LIN {X 0,Y 516.896,Z 484.102,A -85,B 0,C 180,E1 -5072.543,E2 -5072.543} C_VEL
LIN {X 0,Y 516.867,Z 484.105,A -85,B 0,C 180,E1 -5075.329,E2 -5075.329} C_VEL
LIN {X 0,Y 516.881,Z 484.098,A -85,B 0,C 180,E1 -5077.943,E2 -5077.943} C_VEL
LIN {X 0,Y 516.885,Z 484.1,A -85,B 0,C 180,E1 -5080.742,E2 -5080.742} C_VEL
LIN {X 0,Y 516.884,Z 484.103,A -85,B 0,C 180,E1 -5082.831,E2 -5082.831} C_VEL
LIN {X 0,Y 516.897,Z 484.096,A -85,B 0,C 180,E1 -5085.007,E2 -5085.007} C_VEL
LIN {X 0,Y 516.916,Z 484.093,A -85,B 0,C 180,E1 -5088.399,E2 -5088.399} C_VEL
LIN {X 0,Y 516.884,Z 484.143,A -85,B 0,C 180,E1 -5091.046,E2 -5091.046} C_VEL
LIN {X 0,Y 518.914,Z 494.433,A -85,B 0,C 180,E1 -5093.663,E2 -5093.663} C_VEL
LIN {X 0,Y 518.765,Z 503.318,A -85,B 0,C 180,E1 -5095.731,E2 -5095.731} C_VEL
LIN {X 0,Y 518.365,Z 517.844,A -85,B 0,C 180,E1 -5098.989,E2 -5098.989} C_VEL
LIN {X 0,Y 518.058,Z 531.109,A -85,B 0,C 180,E1 -5101.86,E2 -5101.86} C_VEL
LIN {X 0,Y 517.746,Z 545.538,A -85,B 0,C 180,E1 -5104.9,E2 -5104.9} C_VEL
LIN {X 0,Y 517.484,Z 558.916,A -85,B 0,C 180,E1 -5107.65,E2 -5107.65} C_VEL
LIN {X 0,Y 517.263,Z 573.383,A -85,B 0,C 180,E1 -5110.556,E2 -5110.556} C_VEL
LIN {X 0,Y 517.038,Z 587.913,A -85,B 0,C 180,E1 -5113.414,E2 -5113.414} C_VEL
LIN {X 0,Y 516.818,Z 601.396,A -85,B 0,C 180,E1 -5116.057,E2 -5116.057} C_VEL
LIN {X 0,Y 518.532,Z 613.647,A -85,B 0,C 180,E1 -5116.354,E2 -5116.354} C_VEL
LIN {X 0,Y 518.297,Z 626.806,A -85,B 0,C 180,E1 -5116.772,E2 -5116.772} C_VEL
LIN {X 0,Y 518.011,Z 637.948,A -85,B 0,C 180,E1 -5117.263,E2 -5117.263} C_VEL
LIN {X 0,Y 517.786,Z 649.556,A -85,B 0,C 180,E1 -5117.927,E2 -5117.927} C_VEL
LIN {X 0,Y 517.451,Z 660.748,A -85,B 0,C 180,E1 -5118.741,E2 -5118.741} C_VEL
LIN {X 0,Y 517.174,Z 670.566,A -85,B 0,C 180,E1 -5119.627,E2 -5119.627} C_VEL
LIN {X 0,Y 516.898,Z 679.413,A -85,B 0,C 180,E1 -5120.61,E2 -5120.61} C_VEL
LIN {X 0,Y 516.682,Z 688.004,A -85,B 0,C 180,E1 -5121.789,E2 -5121.789} C_VEL
LIN {X 0,Y 516.506,Z 694.868,A -85,B 0,C 180,E1 -5122.966,E2 -5122.966} C_VEL
LIN {X 0,Y 516.454,Z 700.366,A -85,B 0,C 180,E1 -5124.142,E2 -5124.142} C_VEL
LIN {X 0,Y 516.271,Z 704.677,A -85,B 0,C 180,E1 -5125.315,E2 -5125.315} C_VEL
LIN {X 0,Y 516.355,Z 706.958,A -85,B 0,C 180,E1 -5126.098,E2 -5126.098} C_VEL
LIN {X 0,Y 516.282,Z 708.807,A -85,B 0,C 180,E1 -5126.879,E2 -5126.879} C_VEL
LIN {X 0,Y 516.261,Z 710.193,A -85,B 0,C 180,E1 -5127.659,E2 -5127.659} C_VEL
LIN {X 0,Y 516.16,Z 711.785,A -85,B 0,C 180,E1 -5129.22,E2 -5129.22} C_VEL
LIN {X 0,Y 516.154,Z 712,A -85,B 0,C 180,E1 -5130,E2 -5130} C_VEL
LIN {X 0,Y 516.192,Z 711.183,A -85,B 0,C 180,E1 -5131.56,E2 -5131.56} C_VEL
LIN {X 0,Y 516.261,Z 710.196,A -85,B 0,C 180,E1 -5132.341,E2 -5132.341} C_VEL
LIN {X 0,Y 516.282,Z 708.81,A -85,B 0,C 180,E1 -5133.121,E2 -5133.121} C_VEL
LIN {X 0,Y 516.344,Z 705.895,A -85,B 0,C 180,E1 -5134.293,E2 -5134.293} C_VEL
LIN {X 0,Y 516.405,Z 701.947,A -85,B 0,C 180,E1 -5135.467,E2 -5135.467} C_VEL
LIN {X 0,Y 516.486,Z 696.032,A -85,B 0,C 180,E1 -5136.808,E2 -5136.808} C_VEL
LIN {X 0,Y 516.641,Z 689.234,A -85,B 0,C 180,E1 -5138.015,E2 -5138.015} C_VEL
LIN {X 0,Y 516.868,Z 680.991,A -85,B 0,C 180,E1 -5139.194,E2 -5139.194} C_VEL
LIN {X 0,Y 517.081,Z 672.519,A -85,B 0,C 180,E1 -5140.177,E2 -5140.177} C_VEL
LIN {X 0,Y 517.408,Z 661.937,A -85,B 0,C 180,E1 -5141.161,E2 -5141.161} C_VEL
LIN {X 0,Y 517.723,Z 650.028,A -85,B 0,C 180,E1 -5142.04,E2 -5142.04} C_VEL
LIN {X 0,Y 518.043,Z 637.865,A -85,B 0,C 180,E1 -5142.736,E2 -5142.736} C_VEL
LIN {X 0,Y 518.338,Z 625.358,A -85,B 0,C 180,E1 -5143.277,E2 -5143.277} C_VEL
LIN {X 0,Y 518.376,Z 612.02,A -85,B 0,C 180,E1 -5143.688,E2 -5143.688} C_VEL
LIN {X 0,Y 516.818,Z 601.178,A -85,B 0,C 180,E1 -5143.943,E2 -5143.943} C_VEL
LIN {X 0,Y 517.097,Z 584.267,A -85,B 0,C 180,E1 -5147.194,E2 -5147.194} C_VEL
LIN {X 0,Y 517.248,Z 569.103,A -85,B 0,C 180,E1 -5150.113,E2 -5150.113} C_VEL
LIN {X 0,Y 517.442,Z 555.28,A -85,B 0,C 180,E1 -5152.825,E2 -5152.825} C_VEL
LIN {X 0,Y 517.604,Z 541.77,A -85,B 0,C 180,E1 -5155.538,E2 -5155.538} C_VEL
LIN {X 0,Y 517.8,Z 526.86,A -85,B 0,C 180,E1 -5158.584,E2 -5158.584} C_VEL
LIN {X 0,Y 517.993,Z 512.786,A -85,B 0,C 180,E1 -5161.562,E2 -5161.562} C_VEL
LIN {X 0,Y 518.272,Z 498.486,A -85,B 0,C 180,E1 -5164.718,E2 -5164.718} C_VEL
LIN {X 0,Y 518.362,Z 492.293,A -85,B 0,C 180,E1 -5166.142,E2 -5166.142} C_VEL
LIN {X 0,Y 516.897,Z 484.1,A -85,B 0,C 180,E1 -5168.246,E2 -5168.246} C_VEL
LIN {X 0,Y 516.918,Z 484.098,A -85,B 0,C 180,E1 -5171.602,E2 -5171.602} C_VEL
LIN {X 0,Y 516.926,Z 484.1,A -85,B 0,C 180,E1 -5175.01,E2 -5175.01} C_VEL
LIN {X 0,Y 516.919,Z 484.099,A -85,B 0,C 180,E1 -5178.399,E2 -5178.399} C_VEL
LIN {X 0,Y 516.883,Z 484.102,A -85,B 0,C 180,E1 -5181.284,E2 -5181.284} C_VEL
LIN {X 0,Y 516.871,Z 484.102,A -85,B 0,C 180,E1 -5184.22,E2 -5184.22} C_VEL
LIN {X 0,Y 516.884,Z 484.101,A -85,B 0,C 180,E1 -5187.052,E2 -5187.052} C_VEL
LIN {X 0,Y 516.896,Z 484.101,A -85,B 0,C 180,E1 -5189.797,E2 -5189.797} C_VEL
LIN {X 0,Y 516.928,Z 484.096,A -85,B 0,C 180,E1 -5192.467,E2 -5192.467} C_VEL
LIN {X 0,Y 516.876,Z 484.102,A -85,B 0,C 180,E1 -5195.07,E2 -5195.07} C_VEL
LIN {X 0,Y 516.873,Z 484.102,A -85,B 0,C 180,E1 -5197.622,E2 -5197.622} C_VEL
LIN {X 0,Y 516.936,Z 484.095,A -85,B 0,C 180,E1 -5200.13,E2 -5200.13} C_VEL
LIN {X 0,Y 516.91,Z 484.098,A -85,B 0,C 180,E1 -5202.596,E2 -5202.596} C_VEL
LIN {X 0,Y 516.945,Z 484.092,A -85,B 0,C 180,E1 -5205.03,E2 -5205.03} C_VEL
LIN {X 0,Y 516.971,Z 484.09,A -85,B 0,C 180,E1 -5208.234,E2 -5208.234} C_VEL
LIN {X 0,Y 516.969,Z 484.088,A -85,B 0,C 180,E1 -5211.4,E2 -5211.4} C_VEL
LIN {X 0,Y 517.016,Z 484.085,A -85,B 0,C 180,E1 -5213.757,E2 -5213.757} C_VEL
LIN {X 0,Y 517.085,Z 484.075,A -85,B 0,C 180,E1 -5217.663,E2 -5217.663} C_VEL
LIN {X 0,Y 517.097,Z 484.075,A -85,B 0,C 180,E1 -5220.779,E2 -5220.779} C_VEL
LIN {X 0,Y 517.014,Z 484.085,A -85,B 0,C 180,E1 -5223.117,E2 -5223.117} C_VEL
LIN {X 0,Y 516.98,Z 484.088,A -85,B 0,C 180,E1 -5226.244,E2 -5226.244} C_VEL
LIN {X 0,Y 516.97,Z 484.09,A -85,B 0,C 180,E1 -5228.601,E2 -5228.601} C_VEL
LIN {X 0,Y 516.957,Z 484.092,A -85,B 0,C 180,E1 -5231.807,E2 -5231.807} C_VEL
LIN {X 0,Y 516.95,Z 484.093,A -85,B 0,C 180,E1 -5235.147,E2 -5235.147} C_VEL
LIN {X 0,Y 516.922,Z 484.101,A -85,B 0,C 180,E1 -5238.223,E2 -5238.223} C_VEL
LIN {X 0,Y 516.961,Z 484.207,A -85,B 0,C 180,E1 -5240.934,E2 -5240.934} C_VEL
LIN {X 0,Y 518.09,Z 488.502,A -85,B 0,C 180,E1 -5241.173,E2 -5241.173} C_VEL
LIN {X 0,Y 518.099,Z 498.056,A -85,B 0,C 180,E1 -5241.694,E2 -5241.694} C_VEL
LIN {X 0,Y 517.842,Z 508.776,A -85,B 0,C 180,E1 -5242.422,E2 -5242.422} C_VEL
LIN {X 0,Y 517.549,Z 518.004,A -85,B 0,C 180,E1 -5243.192,E2 -5243.192} C_VEL
LIN {X 0,Y 517.283,Z 526.537,A -85,B 0,C 180,E1 -5244.054,E2 -5244.054} C_VEL
LIN {X 0,Y 516.981,Z 535.368,A -85,B 0,C 180,E1 -5245.14,E2 -5245.14} C_VEL
LIN {X 0,Y 516.804,Z 543.287,A -85,B 0,C 180,E1 -5246.365,E2 -5246.365} C_VEL
LIN {X 0,Y 516.615,Z 549.379,A -85,B 0,C 180,E1 -5247.551,E2 -5247.551} C_VEL
LIN {X 0,Y 516.501,Z 553.171,A -85,B 0,C 180,E1 -5248.441,E2 -5248.441} C_VEL
LIN {X 0,Y 516.423,Z 557.58,A -85,B 0,C 180,E1 -5249.791,E2 -5249.791} C_VEL
LIN {X 0,Y 516.345,Z 560.715,A -85,B 0,C 180,E1 -5251.146,E2 -5251.146} C_VEL
LIN {X 0,Y 516.265,Z 562.567,A -85,B 0,C 180,E1 -5252.433,E2 -5252.433} C_VEL
LIN {X 0,Y 516.287,Z 563.411,A -85,B 0,C 180,E1 -5253.926,E2 -5253.926} C_VEL
LIN {X 0,Y 516.253,Z 562.97,A -85,B 0,C 180,E1 -5255.233,E2 -5255.233} C_VEL
LIN {X 0,Y 516.3,Z 560.93,A -85,B 0,C 180,E1 -5256.794,E2 -5256.794} C_VEL
LIN {X 0,Y 516.412,Z 558.616,A -85,B 0,C 180,E1 -5257.876,E2 -5257.876} C_VEL
LIN {X 0,Y 516.47,Z 554.854,A -85,B 0,C 180,E1 -5259.136,E2 -5259.136} C_VEL
LIN {X 0,Y 516.54,Z 551.346,A -85,B 0,C 180,E1 -5260.061,E2 -5260.061} C_VEL
LIN {X 0,Y 516.649,Z 546.133,A -85,B 0,C 180,E1 -5261.168,E2 -5261.168} C_VEL
LIN {X 0,Y 516.811,Z 541.161,A -85,B 0,C 180,E1 -5262.048,E2 -5262.048} C_VEL
LIN {X 0,Y 517.041,Z 534.094,A -85,B 0,C 180,E1 -5263.082,E2 -5263.082} C_VEL
LIN {X 0,Y 517.207,Z 527.215,A -85,B 0,C 180,E1 -5263.93,E2 -5263.93} C_VEL
LIN {X 0,Y 517.478,Z 518.829,A -85,B 0,C 180,E1 -5264.792,E2 -5264.792} C_VEL
LIN {X 0,Y 517.631,Z 513.549,A -85,B 0,C 180,E1 -5265.266,E2 -5265.266} C_VEL
LIN {X 0,Y 517.058,Z 507.251,A -85,B 0,C 180,E1 -5265.784,E2 -5265.784} C_VEL
LIN {X 0,Y 515.311,Z 500.945,A -85,B 0,C 180,E1 -5266.275,E2 -5266.275} C_VEL
LIN {X 0,Y 513.049,Z 494.539,A -85,B 0,C 180,E1 -5266.742,E2 -5266.742} C_VEL
LIN {X 0,Y 510.614,Z 487.934,A -85,B 0,C 180,E1 -5267.163,E2 -5267.163} C_VEL
LIN {X 0,Y 509.873,Z 484.974,A -85,B 0,C 180,E1 -5267.337,E2 -5267.337} C_VEL
LIN {X 0,Y 509.842,Z 484.979,A -85,B 0,C 180,E1 -5270.647,E2 -5270.647} C_VEL
LIN {X 0,Y 509.814,Z 484.982,A -85,B 0,C 180,E1 -5273.646,E2 -5273.646} C_VEL
LIN {X 0,Y 509.864,Z 484.974,A -85,B 0,C 180,E1 -5276.539,E2 -5276.539} C_VEL
LIN {X 0,Y 509.846,Z 484.976,A -85,B 0,C 180,E1 -5279.334,E2 -5279.334} C_VEL
LIN {X 0,Y 509.891,Z 484.97,A -85,B 0,C 180,E1 -5282.054,E2 -5282.054} C_VEL
LIN {X 0,Y 509.823,Z 484.981,A -85,B 0,C 180,E1 -5284.701,E2 -5284.701} C_VEL
LIN {X 0,Y 509.832,Z 484.982,A -85,B 0,C 180,E1 -5287.458,E2 -5287.458} C_VEL
LIN {X 0,Y 509.922,Z 484.967,A -85,B 0,C 180,E1 -5289.845,E2 -5289.845} C_VEL
LIN {X 0,Y 509.872,Z 484.975,A -85,B 0,C 180,E1 -5293.174,E2 -5293.174} C_VEL
LIN {X 0,Y 509.863,Z 484.974,A -85,B 0,C 180,E1 -5295.634,E2 -5295.634} C_VEL
LIN {X 0,Y 509.919,Z 484.967,A -85,B 0,C 180,E1 -5298.874,E2 -5298.874} C_VEL
LIN {X 0,Y 509.915,Z 484.97,A -85,B 0,C 180,E1 -5302.078,E2 -5302.078} C_VEL
LIN {X 0,Y 509.97,Z 484.96,A -85,B 0,C 180,E1 -5304.464,E2 -5304.464} C_VEL
LIN {X 0,Y 510.06,Z 484.949,A -85,B 0,C 180,E1 -5307.631,E2 -5307.631} C_VEL
LIN {X 0,Y 510.067,Z 484.948,A -85,B 0,C 180,E1 -5310.789,E2 -5310.789} C_VEL
LIN {X 0,Y 509.933,Z 484.967,A -85,B 0,C 180,E1 -5313.16,E2 -5313.16} C_VEL
LIN {X 0,Y 509.927,Z 484.966,A -85,B 0,C 180,E1 -5316.33,E2 -5316.33} C_VEL
LIN {X 0,Y 509.916,Z 484.969,A -85,B 0,C 180,E1 -5318.72,E2 -5318.72} C_VEL
LIN {X 0,Y 509.91,Z 484.97,A -85,B 0,C 180,E1 -5321.931,E2 -5321.931} C_VEL
LIN {X 0,Y 509.9,Z 484.97,A -85,B 0,C 180,E1 -5325.242,E2 -5325.242} C_VEL
LIN {X 0,Y 509.862,Z 484.973,A -85,B 0,C 180,E1 -5328.484,E2 -5328.484} C_VEL
LIN {X 0,Y 509.856,Z 484.978,A -85,B 0,C 180,E1 -5331.001,E2 -5331.001} C_VEL
LIN {X 0,Y 509.824,Z 484.982,A -85,B 0,C 180,E1 -5333.564,E2 -5333.564} C_VEL
LIN {X 0,Y 509.882,Z 484.972,A -85,B 0,C 180,E1 -5336.37,E2 -5336.37} C_VEL
LIN {X 0,Y 509.863,Z 484.977,A -85,B 0,C 180,E1 -5339.726,E2 -5339.726} C_VEL
LIN {X 0,Y 509.871,Z 484.976,A -85,B 0,C 180,E1 -5342.773,E2 -5342.773} C_VEL
LIN {X 0,Y 509.826,Z 484.982,A -85,B 0,C 180,E1 -5345.577,E2 -5345.577} C_VEL
LIN {X 0,Y 509.853,Z 484.975,A -85,B 0,C 180,E1 -5348.338,E2 -5348.338} C_VEL
LIN {X 0,Y 509.836,Z 484.979,A -85,B 0,C 180,E1 -5351.428,E2 -5351.428} C_VEL
LIN {X 0,Y 509.843,Z 484.979,A -85,B 0,C 180,E1 -5354.67,E2 -5354.67} C_VEL
LIN {X 0,Y 509.853,Z 484.976,A -85,B 0,C 180,E1 -5358.104,E2 -5358.104} C_VEL
LIN {X 0,Y 509.849,Z 484.978,A -85,B 0,C 180,E1 -5360.647,E2 -5360.647} C_VEL
LIN {X 0,Y 509.809,Z 484.984,A -85,B 0,C 180,E1 -5363.645,E2 -5363.645} C_VEL
LIN {X 0,Y 509.863,Z 484.976,A -85,B 0,C 180,E1 -5366.539,E2 -5366.539} C_VEL
LIN {X 0,Y 509.849,Z 484.977,A -85,B 0,C 180,E1 -5369.334,E2 -5369.334} C_VEL
LIN {X 0,Y 509.895,Z 484.969,A -85,B 0,C 180,E1 -5372.054,E2 -5372.054} C_VEL
LIN {X 0,Y 509.82,Z 484.98,A -85,B 0,C 180,E1 -5374.701,E2 -5374.701} C_VEL
LIN {X 0,Y 509.83,Z 484.979,A -85,B 0,C 180,E1 -5377.458,E2 -5377.458} C_VEL
LIN {X 0,Y 509.918,Z 484.969,A -85,B 0,C 180,E1 -5379.844,E2 -5379.844} C_VEL
LIN {X 0,Y 509.873,Z 484.976,A -85,B 0,C 180,E1 -5383.174,E2 -5383.174} C_VEL
LIN {X 0,Y 509.862,Z 484.975,A -85,B 0,C 180,E1 -5385.634,E2 -5385.634} C_VEL
LIN {X 0,Y 509.917,Z 484.969,A -85,B 0,C 180,E1 -5388.874,E2 -5388.874} C_VEL
LIN {X 0,Y 509.911,Z 484.97,A -85,B 0,C 180,E1 -5392.078,E2 -5392.078} C_VEL
LIN {X 0,Y 509.975,Z 484.96,A -85,B 0,C 180,E1 -5394.464,E2 -5394.464} C_VEL
LIN {X 0,Y 510.053,Z 484.951,A -85,B 0,C 180,E1 -5397.631,E2 -5397.631} C_VEL
LIN {X 0,Y 510.066,Z 484.95,A -85,B 0,C 180,E1 -5400.789,E2 -5400.789} C_VEL
LIN {X 0,Y 509.919,Z 484.967,A -85,B 0,C 180,E1 -5403.16,E2 -5403.16} C_VEL
LIN {X 0,Y 509.928,Z 484.965,A -85,B 0,C 180,E1 -5406.33,E2 -5406.33} C_VEL
LIN {X 0,Y 509.913,Z 484.971,A -85,B 0,C 180,E1 -5408.72,E2 -5408.72} C_VEL
LIN {X 0,Y 509.955,Z 484.964,A -85,B 0,C 180,E1 -5411.93,E2 -5411.93} C_VEL
LIN {X 0,Y 509.897,Z 484.97,A -85,B 0,C 180,E1 -5415.242,E2 -5415.242} C_VEL
LIN {X 0,Y 509.864,Z 484.974,A -85,B 0,C 180,E1 -5418.484,E2 -5418.484} C_VEL
LIN {X 0,Y 509.852,Z 484.976,A -85,B 0,C 180,E1 -5421.002,E2 -5421.002} C_VEL
LIN {X 0,Y 509.823,Z 484.981,A -85,B 0,C 180,E1 -5423.564,E2 -5423.564} C_VEL
LIN {X 0,Y 509.875,Z 484.974,A -85,B 0,C 180,E1 -5426.37,E2 -5426.37} C_VEL
LIN {X 0,Y 509.86,Z 484.976,A -85,B 0,C 180,E1 -5429.726,E2 -5429.726} C_VEL
LIN {X 0,Y 509.868,Z 484.975,A -85,B 0,C 180,E1 -5432.773,E2 -5432.773} C_VEL
LIN {X 0,Y 509.827,Z 484.981,A -85,B 0,C 180,E1 -5435.578,E2 -5435.578} C_VEL
LIN {X 0,Y 509.85,Z 484.977,A -85,B 0,C 180,E1 -5438.338,E2 -5438.338} C_VEL
LIN {X 0,Y 509.857,Z 484.979,A -85,B 0,C 180,E1 -5441.425,E2 -5441.425} C_VEL
LIN {X 0,Y 509.84,Z 484.977,A -85,B 0,C 180,E1 -5444.67,E2 -5444.67} C_VEL
LIN {X 0,Y 509.856,Z 484.972,A -85,B 0,C 180,E1 -5448.104,E2 -5448.104} C_VEL
LIN {X 0,Y 509.847,Z 485.024,A -85,B 0,C 180,E1 -5450.775,E2 -5450.775} C_VEL
LIN {X 0,Y 511.835,Z 494.949,A -85,B 0,C 180,E1 -5453.346,E2 -5453.346} C_VEL
LIN {X 0,Y 512.044,Z 497.933,A -85,B 0,C 180,E1 -5454.076,E2 -5454.076} C_VEL
LIN {X 0,Y 511.677,Z 509.084,A -85,B 0,C 180,E1 -5456.673,E2 -5456.673} C_VEL
LIN {X 0,Y 511.292,Z 523.821,A -85,B 0,C 180,E1 -5459.994,E2 -5459.994} C_VEL
LIN {X 0,Y 510.931,Z 537.675,A -85,B 0,C 180,E1 -5463.004,E2 -5463.004} C_VEL
LIN {X 0,Y 510.624,Z 552.005,A -85,B 0,C 180,E1 -5466.045,E2 -5466.045} C_VEL
LIN {X 0,Y 510.26,Z 567.756,A -85,B 0,C 180,E1 -5469.297,E2 -5469.297} C_VEL
LIN {X 0,Y 510.057,Z 582.932,A -85,B 0,C 180,E1 -5472.354,E2 -5472.354} C_VEL
LIN {X 0,Y 509.79,Z 599.301,A -85,B 0,C 180,E1 -5475.632,E2 -5475.632} C_VEL
LIN {X 0,Y 509.8,Z 600.447,A -85,B 0,C 180,E1 -5475.862,E2 -5475.862} C_VEL
LIN {X 0,Y 510.811,Z 608.526,A -85,B 0,C 180,E1 -5476.049,E2 -5476.049} C_VEL
LIN {X 0,Y 511.563,Z 615.375,A -85,B 0,C 180,E1 -5476.241,E2 -5476.241} C_VEL
LIN {X 0,Y 511.287,Z 628.315,A -85,B 0,C 180,E1 -5476.689,E2 -5476.689} C_VEL
LIN {X 0,Y 510.934,Z 640.657,A -85,B 0,C 180,E1 -5477.286,E2 -5477.286} C_VEL
LIN {X 0,Y 510.637,Z 651.496,A -85,B 0,C 180,E1 -5477.962,E2 -5477.962} C_VEL
LIN {X 0,Y 510.336,Z 662.111,A -85,B 0,C 180,E1 -5478.783,E2 -5478.783} C_VEL
LIN {X 0,Y 510.061,Z 671.583,A -85,B 0,C 180,E1 -5479.681,E2 -5479.681} C_VEL
LIN {X 0,Y 509.802,Z 680.238,A -85,B 0,C 180,E1 -5480.678,E2 -5480.678} C_VEL
LIN {X 0,Y 509.585,Z 688.692,A -85,B 0,C 180,E1 -5481.873,E2 -5481.873} C_VEL
LIN {X 0,Y 509.42,Z 695.519,A -85,B 0,C 180,E1 -5483.067,E2 -5483.067} C_VEL
LIN {X 0,Y 509.322,Z 701.779,A -85,B 0,C 180,E1 -5484.457,E2 -5484.457} C_VEL
LIN {X 0,Y 509.232,Z 705.811,A -85,B 0,C 180,E1 -5485.647,E2 -5485.647} C_VEL
LIN {X 0,Y 509.2,Z 708.77,A -85,B 0,C 180,E1 -5486.835,E2 -5486.835} C_VEL
LIN {X 0,Y 509.161,Z 710.171,A -85,B 0,C 180,E1 -5487.627,E2 -5487.627} C_VEL
LIN {X 0,Y 509.073,Z 711.774,A -85,B 0,C 180,E1 -5489.209,E2 -5489.209} C_VEL
LIN {X 0,Y 509.065,Z 711.991,A -85,B 0,C 180,E1 -5490,E2 -5490} C_VEL
LIN {X 0,Y 509.112,Z 711.169,A -85,B 0,C 180,E1 -5491.582,E2 -5491.582} C_VEL
LIN {X 0,Y 509.161,Z 710.174,A -85,B 0,C 180,E1 -5492.373,E2 -5492.373} C_VEL
LIN {X 0,Y 509.2,Z 708.774,A -85,B 0,C 180,E1 -5493.165,E2 -5493.165} C_VEL
LIN {X 0,Y 509.232,Z 705.812,A -85,B 0,C 180,E1 -5494.353,E2 -5494.353} C_VEL
LIN {X 0,Y 509.322,Z 701.776,A -85,B 0,C 180,E1 -5495.543,E2 -5495.543} C_VEL
LIN {X 0,Y 509.405,Z 695.97,A -85,B 0,C 180,E1 -5496.844,E2 -5496.844} C_VEL
LIN {X 0,Y 509.585,Z 688.657,A -85,B 0,C 180,E1 -5498.127,E2 -5498.127} C_VEL
LIN {X 0,Y 509.802,Z 680.168,A -85,B 0,C 180,E1 -5499.322,E2 -5499.322} C_VEL
LIN {X 0,Y 510.061,Z 671.474,A -85,B 0,C 180,E1 -5500.319,E2 -5500.319} C_VEL
LIN {X 0,Y 510.364,Z 660.755,A -85,B 0,C 180,E1 -5501.317,E2 -5501.317} C_VEL
LIN {X 0,Y 510.671,Z 649.828,A -85,B 0,C 180,E1 -5502.139,E2 -5502.139} C_VEL
LIN {X 0,Y 511.003,Z 638.603,A -85,B 0,C 180,E1 -5502.813,E2 -5502.813} C_VEL
LIN {X 0,Y 511.319,Z 626.732,A -85,B 0,C 180,E1 -5503.361,E2 -5503.361} C_VEL
LIN {X 0,Y 511.473,Z 613.096,A -85,B 0,C 180,E1 -5503.813,E2 -5503.813} C_VEL
LIN {X 0,Y 509.848,Z 601.602,A -85,B 0,C 180,E1 -5504.099,E2 -5504.099} C_VEL
LIN {X 0,Y 509.791,Z 599.936,A -85,B 0,C 180,E1 -5504.164,E2 -5504.164} C_VEL
LIN {X 0,Y 510.007,Z 584.216,A -85,B 0,C 180,E1 -5507.234,E2 -5507.234} C_VEL
LIN {X 0,Y 510.165,Z 569.301,A -85,B 0,C 180,E1 -5510.145,E2 -5510.145} C_VEL
LIN {X 0,Y 510.385,Z 554.534,A -85,B 0,C 180,E1 -5513.107,E2 -5513.107} C_VEL
LIN {X 0,Y 510.583,Z 540.738,A -85,B 0,C 180,E1 -5515.915,E2 -5515.915} C_VEL
LIN {X 0,Y 510.803,Z 525.911,A -85,B 0,C 180,E1 -5519.012,E2 -5519.012} C_VEL
LIN {X 0,Y 511.056,Z 512.231,A -85,B 0,C 180,E1 -5521.969,E2 -5521.969} C_VEL
LIN {X 0,Y 511.361,Z 497.7,A -85,B 0,C 180,E1 -5525.257,E2 -5525.257} C_VEL
LIN {X 0,Y 511.434,Z 493.605,A -85,B 0,C 180,E1 -5526.221,E2 -5526.221} C_VEL
LIN {X 0,Y 509.849,Z 484.978,A -85,B 0,C 180,E1 -5528.465,E2 -5528.465} C_VEL
LIN {X 0,Y 509.86,Z 484.977,A -85,B 0,C 180,E1 -5531.426,E2 -5531.426} C_VEL
LIN {X 0,Y 509.86,Z 484.979,A -85,B 0,C 180,E1 -5534.668,E2 -5534.668} C_VEL
LIN {X 0,Y 509.861,Z 484.977,A -85,B 0,C 180,E1 -5538.103,E2 -5538.103} C_VEL
LIN {X 0,Y 509.849,Z 484.977,A -85,B 0,C 180,E1 -5540.648,E2 -5540.648} C_VEL
LIN {X 0,Y 509.812,Z 484.983,A -85,B 0,C 180,E1 -5543.646,E2 -5543.646} C_VEL
LIN {X 0,Y 509.845,Z 484.978,A -85,B 0,C 180,E1 -5546.538,E2 -5546.538} C_VEL
LIN {X 0,Y 509.849,Z 484.976,A -85,B 0,C 180,E1 -5549.335,E2 -5549.335} C_VEL
LIN {X 0,Y 509.895,Z 484.971,A -85,B 0,C 180,E1 -5552.055,E2 -5552.055} C_VEL
LIN {X 0,Y 509.842,Z 484.979,A -85,B 0,C 180,E1 -5554.702,E2 -5554.702} C_VEL
LIN {X 0,Y 509.83,Z 484.981,A -85,B 0,C 180,E1 -5557.458,E2 -5557.458} C_VEL
LIN {X 0,Y 509.921,Z 484.969,A -85,B 0,C 180,E1 -5559.845,E2 -5559.845} C_VEL
LIN {X 0,Y 509.877,Z 484.973,A -85,B 0,C 180,E1 -5563.175,E2 -5563.175} C_VEL
LIN {X 0,Y 509.865,Z 484.973,A -85,B 0,C 180,E1 -5565.634,E2 -5565.634} C_VEL
LIN {X 0,Y 509.917,Z 484.968,A -85,B 0,C 180,E1 -5568.875,E2 -5568.875} C_VEL
LIN {X 0,Y 509.955,Z 484.963,A -85,B 0,C 180,E1 -5572.079,E2 -5572.079} C_VEL
LIN {X 0,Y 509.985,Z 484.961,A -85,B 0,C 180,E1 -5574.464,E2 -5574.464} C_VEL
LIN {X 0,Y 510.054,Z 484.951,A -85,B 0,C 180,E1 -5577.631,E2 -5577.631} C_VEL
LIN {X 0,Y 510.068,Z 484.951,A -85,B 0,C 180,E1 -5580.79,E2 -5580.79} C_VEL
LIN {X 0,Y 509.956,Z 484.965,A -85,B 0,C 180,E1 -5583.16,E2 -5583.16} C_VEL
LIN {X 0,Y 509.929,Z 484.966,A -85,B 0,C 180,E1 -5586.33,E2 -5586.33} C_VEL
LIN {X 0,Y 509.916,Z 484.968,A -85,B 0,C 180,E1 -5588.72,E2 -5588.72} C_VEL
LIN {X 0,Y 509.909,Z 484.97,A -85,B 0,C 180,E1 -5591.932,E2 -5591.932} C_VEL
LIN {X 0,Y 509.9,Z 484.971,A -85,B 0,C 180,E1 -5595.242,E2 -5595.242} C_VEL
LIN {X 0,Y 509.866,Z 484.98,A -85,B 0,C 180,E1 -5598.484,E2 -5598.484} C_VEL
LIN {X 0,Y 509.89,Z 484.976,A -85,B 0,C 180,E1 -5600.737,E2 -5600.737} C_VEL
LIN {X 0,Y 511.321,Z 490.39,A -85,B 0,C 180,E1 -5601.044,E2 -5601.044} C_VEL
LIN {X 0,Y 511.17,Z 501.613,A -85,B 0,C 180,E1 -5601.685,E2 -5601.685} C_VEL
LIN {X 0,Y 510.876,Z 512.139,A -85,B 0,C 180,E1 -5602.443,E2 -5602.443} C_VEL
LIN {X 0,Y 510.52,Z 523.02,A -85,B 0,C 180,E1 -5603.424,E2 -5603.424} C_VEL
LIN {X 0,Y 510.215,Z 531.765,A -85,B 0,C 180,E1 -5604.409,E2 -5604.409} C_VEL
LIN {X 0,Y 509.964,Z 539.736,A -85,B 0,C 180,E1 -5605.51,E2 -5605.51} C_VEL
LIN {X 0,Y 509.786,Z 546.495,A -85,B 0,C 180,E1 -5606.661,E2 -5606.661} C_VEL
LIN {X 0,Y 509.598,Z 552.621,A -85,B 0,C 180,E1 -5607.964,E2 -5607.964} C_VEL
LIN {X 0,Y 509.486,Z 557.272,A -85,B 0,C 180,E1 -5609.253,E2 -5609.253} C_VEL
LIN {X 0,Y 509.378,Z 561,A -85,B 0,C 180,E1 -5610.697,E2 -5610.697} C_VEL
LIN {X 0,Y 509.311,Z 562.68,A -85,B 0,C 180,E1 -5611.626,E2 -5611.626} C_VEL
LIN {X 0,Y 509.247,Z 563.871,A -85,B 0,C 180,E1 -5612.664,E2 -5612.664} C_VEL
LIN {X 0,Y 509.268,Z 564.441,A -85,B 0,C 180,E1 -5614.104,E2 -5614.104} C_VEL
LIN {X 0,Y 509.241,Z 563.756,A -85,B 0,C 180,E1 -5615.486,E2 -5615.486} C_VEL
LIN {X 0,Y 509.281,Z 561.942,A -85,B 0,C 180,E1 -5616.832,E2 -5616.832} C_VEL
LIN {X 0,Y 509.403,Z 559.033,A -85,B 0,C 180,E1 -5618.149,E2 -5618.149} C_VEL
LIN {X 0,Y 509.492,Z 555.089,A -85,B 0,C 180,E1 -5619.423,E2 -5619.423} C_VEL
LIN {X 0,Y 509.606,Z 550.033,A -85,B 0,C 180,E1 -5620.667,E2 -5620.667} C_VEL
LIN {X 0,Y 509.757,Z 543.76,A -85,B 0,C 180,E1 -5621.884,E2 -5621.884} C_VEL
LIN {X 0,Y 510.048,Z 535.913,A -85,B 0,C 180,E1 -5623.089,E2 -5623.089} C_VEL
LIN {X 0,Y 510.293,Z 528.222,A -85,B 0,C 180,E1 -5624.055,E2 -5624.055} C_VEL
LIN {X 0,Y 510.6,Z 519.045,A -85,B 0,C 180,E1 -5625.003,E2 -5625.003} C_VEL
LIN {X 0,Y 510.848,Z 509.448,A -85,B 0,C 180,E1 -5625.817,E2 -5625.817} C_VEL
LIN {X 0,Y 511.147,Z 499.759,A -85,B 0,C 180,E1 -5626.486,E2 -5626.486} C_VEL
LIN {X 0,Y 511.31,Z 490.403,A -85,B 0,C 180,E1 -5627.013,E2 -5627.013} C_VEL
LIN {X 0,Y 510.614,Z 487.934,A -85,B 0,C 180,E1 -5627.163,E2 -5627.163} C_VEL
LIN {X 0,Y 509.786,Z 486.26,A -85,B 0,C 180,E1 -5627.355,E2 -5627.355} C_VEL
LIN {X 0,Y 508.475,Z 485.274,A -85,B 0,C 180,E1 -5627.704,E2 -5627.704} C_VEL
LIN {X 0,Y 505.635,Z 485.501,A -85,B 0,C 180,E1 -5628.632,E2 -5628.632} C_VEL
LIN {X 0,Y 503.597,Z 485.897,A -85,B 0,C 180,E1 -5629.602,E2 -5629.602} C_VEL
LIN {X 0,Y 502.779,Z 485.857,A -85,B 0,C 180,E1 -5630.597,E2 -5630.597} C_VEL
LIN {X 0,Y 502.759,Z 485.859,A -85,B 0,C 180,E1 -5633.052,E2 -5633.052} C_VEL
LIN {X 0,Y 502.808,Z 485.852,A -85,B 0,C 180,E1 -5636.006,E2 -5636.006} C_VEL
LIN {X 0,Y 502.799,Z 485.855,A -85,B 0,C 180,E1 -5638.857,E2 -5638.857} C_VEL
LIN {X 0,Y 502.846,Z 485.849,A -85,B 0,C 180,E1 -5641.706,E2 -5641.706} C_VEL
LIN {X 0,Y 502.804,Z 485.855,A -85,B 0,C 180,E1 -5644.322,E2 -5644.322} C_VEL
LIN {X 0,Y 502.809,Z 485.856,A -85,B 0,C 180,E1 -5647.298,E2 -5647.298} C_VEL
LIN {X 0,Y 502.825,Z 485.853,A -85,B 0,C 180,E1 -5650.4,E2 -5650.4} C_VEL
LIN {X 0,Y 502.817,Z 485.852,A -85,B 0,C 180,E1 -5652.931,E2 -5652.931} C_VEL
LIN {X 0,Y 502.846,Z 485.849,A -85,B 0,C 180,E1 -5655.429,E2 -5655.429} C_VEL
LIN {X 0,Y 502.883,Z 485.843,A -85,B 0,C 180,E1 -5658.717,E2 -5658.717} C_VEL
LIN {X 0,Y 502.878,Z 485.845,A -85,B 0,C 180,E1 -5661.966,E2 -5661.966} C_VEL
LIN {X 0,Y 502.923,Z 485.838,A -85,B 0,C 180,E1 -5664.386,E2 -5664.386} C_VEL
LIN {X 0,Y 503.03,Z 485.825,A -85,B 0,C 180,E1 -5667.598,E2 -5667.598} C_VEL
LIN {X 0,Y 503.016,Z 485.827,A -85,B 0,C 180,E1 -5670.8,E2 -5670.8} C_VEL
LIN {X 0,Y 503.026,Z 485.825,A -85,B 0,C 180,E1 -5672.402,E2 -5672.402} C_VEL
LIN {X 0,Y 502.921,Z 485.842,A -85,B 0,C 180,E1 -5675.614,E2 -5675.614} C_VEL
LIN {X 0,Y 502.875,Z 485.848,A -85,B 0,C 180,E1 -5678.843,E2 -5678.843} C_VEL
LIN {X 0,Y 502.851,Z 485.848,A -85,B 0,C 180,E1 -5682.101,E2 -5682.101} C_VEL
LIN {X 0,Y 502.854,Z 485.847,A -85,B 0,C 180,E1 -5685.4,E2 -5685.4} C_VEL
LIN {X 0,Y 502.828,Z 485.85,A -85,B 0,C 180,E1 -5688.752,E2 -5688.752} C_VEL
LIN {X 0,Y 502.789,Z 485.856,A -85,B 0,C 180,E1 -5691.311,E2 -5691.311} C_VEL
LIN {X 0,Y 502.774,Z 485.859,A -85,B 0,C 180,E1 -5693.915,E2 -5693.915} C_VEL
LIN {X 0,Y 502.84,Z 485.85,A -85,B 0,C 180,E1 -5696.568,E2 -5696.568} C_VEL
LIN {X 0,Y 502.819,Z 485.853,A -85,B 0,C 180,E1 -5699.935,E2 -5699.935} C_VEL
LIN {X 0,Y 502.834,Z 485.852,A -85,B 0,C 180,E1 -5703.031,E2 -5703.031} C_VEL
LIN {X 0,Y 502.771,Z 485.859,A -85,B 0,C 180,E1 -5705.951,E2 -5705.951} C_VEL
LIN {X 0,Y 502.798,Z 485.857,A -85,B 0,C 180,E1 -5708.977,E2 -5708.977} C_VEL
LIN {X 0,Y 502.774,Z 485.857,A -85,B 0,C 180,E1 -5712.195,E2 -5712.195} C_VEL
LIN {X 0,Y 502.789,Z 485.855,A -85,B 0,C 180,E1 -5715.47,E2 -5715.47} C_VEL
LIN {X 0,Y 502.798,Z 485.856,A -85,B 0,C 180,E1 -5717.86,E2 -5717.86} C_VEL
LIN {X 0,Y 502.804,Z 485.855,A -85,B 0,C 180,E1 -5721.024,E2 -5721.024} C_VEL
LIN {X 0,Y 502.773,Z 485.857,A -85,B 0,C 180,E1 -5724.17,E2 -5724.17} C_VEL
LIN {X 0,Y 502.836,Z 485.851,A -85,B 0,C 180,E1 -5726.993,E2 -5726.993} C_VEL
LIN {X 0,Y 502.819,Z 485.852,A -85,B 0,C 180,E1 -5730.065,E2 -5730.065} C_VEL
LIN {X 0,Y 502.831,Z 485.851,A -85,B 0,C 180,E1 -5732.533,E2 -5732.533} C_VEL
LIN {X 0,Y 502.784,Z 485.858,A -85,B 0,C 180,E1 -5735.31,E2 -5735.31} C_VEL
LIN {X 0,Y 502.783,Z 485.854,A -85,B 0,C 180,E1 -5737.826,E2 -5737.826} C_VEL
LIN {X 0,Y 502.823,Z 485.854,A -85,B 0,C 180,E1 -5740.4,E2 -5740.4} C_VEL
LIN {X 0,Y 502.818,Z 485.854,A -85,B 0,C 180,E1 -5742.931,E2 -5742.931} C_VEL
LIN {X 0,Y 502.845,Z 485.848,A -85,B 0,C 180,E1 -5745.429,E2 -5745.429} C_VEL
LIN {X 0,Y 502.881,Z 485.844,A -85,B 0,C 180,E1 -5748.717,E2 -5748.717} C_VEL
LIN {X 0,Y 502.875,Z 485.846,A -85,B 0,C 180,E1 -5751.966,E2 -5751.966} C_VEL
LIN {X 0,Y 502.928,Z 485.837,A -85,B 0,C 180,E1 -5754.386,E2 -5754.386} C_VEL
LIN {X 0,Y 503.022,Z 485.827,A -85,B 0,C 180,E1 -5757.598,E2 -5757.598} C_VEL
LIN {X 0,Y 503.036,Z 485.826,A -85,B 0,C 180,E1 -5760.8,E2 -5760.8} C_VEL
LIN {X 0,Y 502.863,Z 485.846,A -85,B 0,C 180,E1 -5763.205,E2 -5763.205} C_VEL
LIN {X 0,Y 502.88,Z 485.844,A -85,B 0,C 180,E1 -5766.419,E2 -5766.419} C_VEL
LIN {X 0,Y 502.871,Z 485.847,A -85,B 0,C 180,E1 -5768.843,E2 -5768.843} C_VEL
LIN {X 0,Y 502.897,Z 485.842,A -85,B 0,C 180,E1 -5772.1,E2 -5772.1} C_VEL
LIN {X 0,Y 502.851,Z 485.847,A -85,B 0,C 180,E1 -5775.4,E2 -5775.4} C_VEL
LIN {X 0,Y 502.829,Z 485.852,A -85,B 0,C 180,E1 -5778.752,E2 -5778.752} C_VEL
LIN {X 0,Y 502.785,Z 485.855,A -85,B 0,C 180,E1 -5781.311,E2 -5781.311} C_VEL
LIN {X 0,Y 502.775,Z 485.858,A -85,B 0,C 180,E1 -5783.914,E2 -5783.914} C_VEL
LIN {X 0,Y 502.836,Z 485.853,A -85,B 0,C 180,E1 -5786.568,E2 -5786.568} C_VEL
LIN {X 0,Y 502.817,Z 485.852,A -85,B 0,C 180,E1 -5789.935,E2 -5789.935} C_VEL
LIN {X 0,Y 502.831,Z 485.85,A -85,B 0,C 180,E1 -5793.031,E2 -5793.031} C_VEL
LIN {X 0,Y 502.775,Z 485.858,A -85,B 0,C 180,E1 -5795.951,E2 -5795.951} C_VEL
LIN {X 0,Y 502.798,Z 485.855,A -85,B 0,C 180,E1 -5798.976,E2 -5798.976} C_VEL
LIN {X 0,Y 502.797,Z 485.854,A -85,B 0,C 180,E1 -5802.139,E2 -5802.139} C_VEL
LIN {X 0,Y 502.787,Z 485.854,A -85,B 0,C 180,E1 -5805.47,E2 -5805.47} C_VEL
LIN {X 0,Y 502.822,Z 485.851,A -85,B 0,C 180,E1 -5808.934,E2 -5808.934} C_VEL
LIN {X 0,Y 502.82,Z 485.946,A -85,B 0,C 180,E1 -5810.509,E2 -5810.509} C_VEL
LIN {X 0,Y 504.869,Z 496.273,A -85,B 0,C 180,E1 -5813.232,E2 -5813.232} C_VEL
LIN {X 0,Y 505.121,Z 500.364,A -85,B 0,C 180,E1 -5814.242,E2 -5814.242} C_VEL
LIN {X 0,Y 504.63,Z 513.55,A -85,B 0,C 180,E1 -5817.339,E2 -5817.339} C_VEL
LIN {X 0,Y 504.236,Z 526.753,A -85,B 0,C 180,E1 -5820.344,E2 -5820.344} C_VEL
LIN {X 0,Y 503.848,Z 541.046,A -85,B 0,C 180,E1 -5823.49,E2 -5823.49} C_VEL
LIN {X 0,Y 503.527,Z 554.354,A -85,B 0,C 180,E1 -5826.342,E2 -5826.342} C_VEL
LIN {X 0,Y 503.182,Z 569.678,A -85,B 0,C 180,E1 -5829.563,E2 -5829.563} C_VEL
LIN {X 0,Y 502.98,Z 584.023,A -85,B 0,C 180,E1 -5832.518,E2 -5832.518} C_VEL
LIN {X 0,Y 502.691,Z 599.486,A -85,B 0,C 180,E1 -5835.657,E2 -5835.657} C_VEL
LIN {X 0,Y 503.928,Z 609.733,A -85,B 0,C 180,E1 -5835.906,E2 -5835.906} C_VEL
LIN {X 0,Y 504.609,Z 616.101,A -85,B 0,C 180,E1 -5836.099,E2 -5836.099} C_VEL
LIN {X 0,Y 504.306,Z 628.425,A -85,B 0,C 180,E1 -5836.552,E2 -5836.552} C_VEL
LIN {X 0,Y 503.908,Z 641.206,A -85,B 0,C 180,E1 -5837.196,E2 -5837.196} C_VEL
LIN {X 0,Y 503.598,Z 652.246,A -85,B 0,C 180,E1 -5837.917,E2 -5837.917} C_VEL
LIN {X 0,Y 503.243,Z 663.346,A -85,B 0,C 180,E1 -5838.827,E2 -5838.827} C_VEL
LIN {X 0,Y 502.934,Z 672.402,A -85,B 0,C 180,E1 -5839.737,E2 -5839.737} C_VEL
LIN {X 0,Y 502.673,Z 682.264,A -85,B 0,C 180,E1 -5840.95,E2 -5840.95} C_VEL
LIN {X 0,Y 502.454,Z 690.138,A -85,B 0,C 180,E1 -5842.162,E2 -5842.162} C_VEL
LIN {X 0,Y 502.275,Z 697.399,A -85,B 0,C 180,E1 -5843.573,E2 -5843.573} C_VEL
LIN {X 0,Y 502.21,Z 702.243,A -85,B 0,C 180,E1 -5844.781,E2 -5844.781} C_VEL
LIN {X 0,Y 502.187,Z 705.951,A -85,B 0,C 180,E1 -5845.988,E2 -5845.988} C_VEL
LIN {X 0,Y 502.152,Z 707.859,A -85,B 0,C 180,E1 -5846.791,E2 -5846.791} C_VEL
LIN {X 0,Y 502.107,Z 709.289,A -85,B 0,C 180,E1 -5847.593,E2 -5847.593} C_VEL
LIN {X 0,Y 502.061,Z 710.306,A -85,B 0,C 180,E1 -5848.396,E2 -5848.396} C_VEL
LIN {X 0,Y 502.024,Z 710.925,A -85,B 0,C 180,E1 -5849.198,E2 -5849.198} C_VEL
LIN {X 0,Y 502.017,Z 711.142,A -85,B 0,C 180,E1 -5850,E2 -5850} C_VEL
LIN {X 0,Y 502.024,Z 710.918,A -85,B 0,C 180,E1 -5850.802,E2 -5850.802} C_VEL
LIN {X 0,Y 502.063,Z 710.296,A -85,B 0,C 180,E1 -5851.604,E2 -5851.604} C_VEL
LIN {X 0,Y 502.109,Z 709.274,A -85,B 0,C 180,E1 -5852.407,E2 -5852.407} C_VEL
LIN {X 0,Y 502.152,Z 707.834,A -85,B 0,C 180,E1 -5853.209,E2 -5853.209} C_VEL
LIN {X 0,Y 502.167,Z 704.802,A -85,B 0,C 180,E1 -5854.415,E2 -5854.415} C_VEL
LIN {X 0,Y 502.265,Z 700.711,A -85,B 0,C 180,E1 -5855.621,E2 -5855.621} C_VEL
LIN {X 0,Y 502.333,Z 694.51,A -85,B 0,C 180,E1 -5857.012,E2 -5857.012} C_VEL
LIN {X 0,Y 502.542,Z 687.546,A -85,B 0,C 180,E1 -5858.242,E2 -5858.242} C_VEL
LIN {X 0,Y 502.747,Z 679.029,A -85,B 0,C 180,E1 -5859.454,E2 -5859.454} C_VEL
LIN {X 0,Y 503.072,Z 669.32,A -85,B 0,C 180,E1 -5860.566,E2 -5860.566} C_VEL
LIN {X 0,Y 503.392,Z 658.377,A -85,B 0,C 180,E1 -5861.578,E2 -5861.578} C_VEL
LIN {X 0,Y 503.689,Z 646.823,A -85,B 0,C 180,E1 -5862.433,E2 -5862.433} C_VEL
LIN {X 0,Y 504.076,Z 634.387,A -85,B 0,C 180,E1 -5863.146,E2 -5863.146} C_VEL
LIN {X 0,Y 504.418,Z 621.549,A -85,B 0,C 180,E1 -5863.701,E2 -5863.701} C_VEL
LIN {X 0,Y 504.418,Z 613.184,A -85,B 0,C 180,E1 -5863.971,E2 -5863.971} C_VEL
LIN {X 0,Y 502.956,Z 602.569,A -85,B 0,C 180,E1 -5864.258,E2 -5864.258} C_VEL
LIN {X 0,Y 502.677,Z 598.88,A -85,B 0,C 180,E1 -5864.343,E2 -5864.343} C_VEL
LIN {X 0,Y 502.945,Z 583.109,A -85,B 0,C 180,E1 -5867.484,E2 -5867.484} C_VEL
LIN {X 0,Y 503.129,Z 567.288,A -85,B 0,C 180,E1 -5870.626,E2 -5870.626} C_VEL
LIN {X 0,Y 503.358,Z 552.43,A -85,B 0,C 180,E1 -5873.667,E2 -5873.667} C_VEL
LIN {X 0,Y 503.602,Z 538.678,A -85,B 0,C 180,E1 -5876.524,E2 -5876.524} C_VEL
LIN {X 0,Y 503.813,Z 523.909,A -85,B 0,C 180,E1 -5879.684,E2 -5879.684} C_VEL
LIN {X 0,Y 504.104,Z 511.374,A -85,B 0,C 180,E1 -5882.463,E2 -5882.463} C_VEL
LIN {X 0,Y 504.522,Z 496.955,A -85,B 0,C 180,E1 -5885.808,E2 -5885.808} C_VEL
LIN {X 0,Y 504.161,Z 492.852,A -85,B 0,C 180,E1 -5886.829,E2 -5886.829} C_VEL
LIN {X 0,Y 502.813,Z 485.855,A -85,B 0,C 180,E1 -5888.697,E2 -5888.697} C_VEL
LIN {X 0,Y 502.823,Z 485.852,A -85,B 0,C 180,E1 -5891.066,E2 -5891.066} C_VEL
LIN {X 0,Y 502.804,Z 485.857,A -85,B 0,C 180,E1 -5894.532,E2 -5894.532} C_VEL
LIN {X 0,Y 502.8,Z 485.857,A -85,B 0,C 180,E1 -5897.861,E2 -5897.861} C_VEL
LIN {X 0,Y 502.804,Z 485.857,A -85,B 0,C 180,E1 -5901.024,E2 -5901.024} C_VEL
LIN {X 0,Y 502.774,Z 485.858,A -85,B 0,C 180,E1 -5904.17,E2 -5904.17} C_VEL
LIN {X 0,Y 502.834,Z 485.851,A -85,B 0,C 180,E1 -5906.994,E2 -5906.994} C_VEL
LIN {X 0,Y 502.819,Z 485.852,A -85,B 0,C 180,E1 -5910.065,E2 -5910.065} C_VEL
LIN {X 0,Y 502.835,Z 485.85,A -85,B 0,C 180,E1 -5912.533,E2 -5912.533} C_VEL
LIN {X 0,Y 502.806,Z 485.853,A -85,B 0,C 180,E1 -5915.305,E2 -5915.305} C_VEL
LIN {X 0,Y 502.784,Z 485.856,A -85,B 0,C 180,E1 -5917.827,E2 -5917.827} C_VEL
LIN {X 0,Y 502.828,Z 485.851,A -85,B 0,C 180,E1 -5920.4,E2 -5920.4} C_VEL
LIN {X 0,Y 502.822,Z 485.851,A -85,B 0,C 180,E1 -5922.931,E2 -5922.931} C_VEL
LIN {X 0,Y 502.847,Z 485.846,A -85,B 0,C 180,E1 -5925.429,E2 -5925.429} C_VEL
LIN {X 0,Y 502.881,Z 485.845,A -85,B 0,C 180,E1 -5928.717,E2 -5928.717} C_VEL
LIN {X 0,Y 502.905,Z 485.84,A -85,B 0,C 180,E1 -5931.967,E2 -5931.967} C_VEL
LIN {X 0,Y 502.942,Z 485.838,A -85,B 0,C 180,E1 -5934.387,E2 -5934.387} C_VEL
LIN {X 0,Y 503.023,Z 485.827,A -85,B 0,C 180,E1 -5937.598,E2 -5937.598} C_VEL
LIN {X 0,Y 503.038,Z 485.827,A -85,B 0,C 180,E1 -5940.801,E2 -5940.801} C_VEL
LIN {X 0,Y 502.9,Z 485.844,A -85,B 0,C 180,E1 -5943.205,E2 -5943.205} C_VEL
LIN {X 0,Y 502.881,Z 485.844,A -85,B 0,C 180,E1 -5946.42,E2 -5946.42} C_VEL
LIN {X 0,Y 502.875,Z 485.845,A -85,B 0,C 180,E1 -5948.844,E2 -5948.844} C_VEL
LIN {X 0,Y 502.85,Z 485.851,A -85,B 0,C 180,E1 -5952.102,E2 -5952.102} C_VEL
LIN {X 0,Y 502.854,Z 485.849,A -85,B 0,C 180,E1 -5955.4,E2 -5955.4} C_VEL
LIN {X 0,Y 502.832,Z 485.856,A -85,B 0,C 180,E1 -5958.752,E2 -5958.752} C_VEL
LIN {X 0,Y 502.85,Z 485.856,A -85,B 0,C 180,E1 -5960.541,E2 -5960.541} C_VEL
LIN {X 0,Y 504.555,Z 492.881,A -85,B 0,C 180,E1 -5960.944,E2 -5960.944} C_VEL
LIN {X 0,Y 504.252,Z 505.102,A -85,B 0,C 180,E1 -5961.675,E2 -5961.675} C_VEL
LIN {X 0,Y 503.902,Z 516.403,A -85,B 0,C 180,E1 -5962.554,E2 -5962.554} C_VEL
LIN {X 0,Y 503.536,Z 526.603,A -85,B 0,C 180,E1 -5963.549,E2 -5963.549} C_VEL
LIN {X 0,Y 503.257,Z 534.902,A -85,B 0,C 180,E1 -5964.549,E2 -5964.549} C_VEL
LIN {X 0,Y 502.973,Z 542.547,A -85,B 0,C 180,E1 -5965.669,E2 -5965.669} C_VEL
LIN {X 0,Y 502.77,Z 549.887,A -85,B 0,C 180,E1 -5967.021,E2 -5967.021} C_VEL
LIN {X 0,Y 502.531,Z 555.647,A -85,B 0,C 180,E1 -5968.392,E2 -5968.392} C_VEL
LIN {X 0,Y 502.434,Z 560.169,A -85,B 0,C 180,E1 -5969.859,E2 -5969.859} C_VEL
LIN {X 0,Y 502.316,Z 563.418,A -85,B 0,C 180,E1 -5971.409,E2 -5971.409} C_VEL
LIN {X 0,Y 502.222,Z 565.19,A -85,B 0,C 180,E1 -5973.077,E2 -5973.077} C_VEL
LIN {X 0,Y 502.227,Z 565.406,A -85,B 0,C 180,E1 -5974.347,E2 -5974.347} C_VEL
LIN {X 0,Y 502.213,Z 564.526,A -85,B 0,C 180,E1 -5975.741,E2 -5975.741} C_VEL
LIN {X 0,Y 502.307,Z 562.515,A -85,B 0,C 180,E1 -5977.106,E2 -5977.106} C_VEL
LIN {X 0,Y 502.397,Z 559.453,A -85,B 0,C 180,E1 -5978.428,E2 -5978.428} C_VEL
LIN {X 0,Y 502.518,Z 555.312,A -85,B 0,C 180,E1 -5979.717,E2 -5979.717} C_VEL
LIN {X 0,Y 502.691,Z 549.508,A -85,B 0,C 180,E1 -5981.079,E2 -5981.079} C_VEL
LIN {X 0,Y 502.904,Z 542.262,A -85,B 0,C 180,E1 -5982.399,E2 -5982.399} C_VEL
LIN {X 0,Y 503.222,Z 534.189,A -85,B 0,C 180,E1 -5983.569,E2 -5983.569} C_VEL
LIN {X 0,Y 503.515,Z 525.375,A -85,B 0,C 180,E1 -5984.614,E2 -5984.614} C_VEL
LIN {X 0,Y 503.893,Z 513.995,A -85,B 0,C 180,E1 -5985.691,E2 -5985.691} C_VEL
LIN {X 0,Y 504.19,Z 503.782,A -85,B 0,C 180,E1 -5986.456,E2 -5986.456} C_VEL
LIN {X 0,Y 504.485,Z 493.25,A -85,B 0,C 180,E1 -5987.087,E2 -5987.087} C_VEL
LIN {X 0,Y 503.978,Z 490.212,A -85,B 0,C 180,E1 -5987.263,E2 -5987.263} C_VEL
LIN {X 0,Y 502.809,Z 485.855,A -85,B 0,C 180,E1 -5987.524,E2 -5987.524} C_VEL
LIN {X 0,Y 502.779,Z 485.857,A -85,B 0,C 180,E1 -5990.597,E2 -5990.597} C_VEL
LIN {X 0,Y 502.12,Z 485.943,A -85,B 0,C 180,E1 -5991.265,E2 -5991.265} C_VEL
LIN {X 0,Y 499.244,Z 486.303,A -85,B 0,C 180,E1 -5992.35,E2 -5992.35} C_VEL
LIN {X 0,Y 496.818,Z 486.604,A -85,B 0,C 180,E1 -5993.224,E2 -5993.224} C_VEL
LIN {X 0,Y 495.796,Z 486.729,A -85,B 0,C 180,E1 -5993.899,E2 -5993.899} C_VEL
LIN {X 0,Y 495.725,Z 486.736,A -85,B 0,C 180,E1 -5994.128,E2 -5994.128} C_VEL
LIN {X 0,Y 495.798,Z 486.727,A -85,B 0,C 180,E1 -5996.756,E2 -5996.756} C_VEL
LIN {X 0,Y 495.768,Z 486.733,A -85,B 0,C 180,E1 -5999.853,E2 -5999.853} C_VEL
LIN {X 0,Y 495.781,Z 486.727,A -85,B 0,C 180,E1 -6002.108,E2 -6002.108} C_VEL
LIN {X 0,Y 495.74,Z 486.735,A -85,B 0,C 180,E1 -6004.83,E2 -6004.83} C_VEL
LIN {X 0,Y 495.754,Z 486.735,A -85,B 0,C 180,E1 -6007.495,E2 -6007.495} C_VEL
LIN {X 0,Y 495.774,Z 486.731,A -85,B 0,C 180,E1 -6010.11,E2 -6010.11} C_VEL
LIN {X 0,Y 495.763,Z 486.73,A -85,B 0,C 180,E1 -6012.68,E2 -6012.68} C_VEL
LIN {X 0,Y 495.793,Z 486.729,A -85,B 0,C 180,E1 -6015.217,E2 -6015.217} C_VEL
LIN {X 0,Y 495.858,Z 486.718,A -85,B 0,C 180,E1 -6018.555,E2 -6018.555} C_VEL
LIN {X 0,Y 495.837,Z 486.722,A -85,B 0,C 180,E1 -6021.851,E2 -6021.851} C_VEL
LIN {X 0,Y 495.84,Z 486.722,A -85,B 0,C 180,E1 -6025.121,E2 -6025.121} C_VEL
LIN {X 0,Y 495.999,Z 486.701,A -85,B 0,C 180,E1 -6027.564,E2 -6027.564} C_VEL
LIN {X 0,Y 495.968,Z 486.705,A -85,B 0,C 180,E1 -6030.812,E2 -6030.812} C_VEL
LIN {X 0,Y 495.994,Z 486.702,A -85,B 0,C 180,E1 -6032.436,E2 -6032.436} C_VEL
LIN {X 0,Y 495.876,Z 486.72,A -85,B 0,C 180,E1 -6035.694,E2 -6035.694} C_VEL
LIN {X 0,Y 495.843,Z 486.724,A -85,B 0,C 180,E1 -6038.97,E2 -6038.97} C_VEL
LIN {X 0,Y 495.834,Z 486.723,A -85,B 0,C 180,E1 -6042.035,E2 -6042.035} C_VEL
LIN {X 0,Y 495.829,Z 486.722,A -85,B 0,C 180,E1 -6045.451,E2 -6045.451} C_VEL
LIN {X 0,Y 495.784,Z 486.729,A -85,B 0,C 180,E1 -6049.028,E2 -6049.028} C_VEL
LIN {X 0,Y 495.748,Z 486.732,A -85,B 0,C 180,E1 -6051.629,E2 -6051.629} C_VEL
LIN {X 0,Y 495.721,Z 486.736,A -85,B 0,C 180,E1 -6054.277,E2 -6054.277} C_VEL
LIN {X 0,Y 495.765,Z 486.733,A -85,B 0,C 180,E1 -6056.977,E2 -6056.977} C_VEL
LIN {X 0,Y 495.768,Z 486.73,A -85,B 0,C 180,E1 -6060.147,E2 -6060.147} C_VEL
LIN {X 0,Y 495.793,Z 486.727,A -85,B 0,C 180,E1 -6063.243,E2 -6063.243} C_VEL
LIN {X 0,Y 495.716,Z 486.737,A -85,B 0,C 180,E1 -6066.087,E2 -6066.087} C_VEL
LIN {X 0,Y 495.762,Z 486.734,A -85,B 0,C 180,E1 -6068.767,E2 -6068.767} C_VEL
LIN {X 0,Y 495.747,Z 486.734,A -85,B 0,C 180,E1 -6071.782,E2 -6071.782} C_VEL
LIN {X 0,Y 495.741,Z 486.734,A -85,B 0,C 180,E1 -6075.141,E2 -6075.141} C_VEL
LIN {X 0,Y 495.754,Z 486.732,A -85,B 0,C 180,E1 -6078.218,E2 -6078.218} C_VEL
LIN {X 0,Y 495.752,Z 486.732,A -85,B 0,C 180,E1 -6081.408,E2 -6081.408} C_VEL
LIN {X 0,Y 495.748,Z 486.732,A -85,B 0,C 180,E1 -6084.462,E2 -6084.462} C_VEL
LIN {X 0,Y 495.771,Z 486.729,A -85,B 0,C 180,E1 -6087.405,E2 -6087.405} C_VEL
LIN {X 0,Y 495.77,Z 486.729,A -85,B 0,C 180,E1 -6090.253,E2 -6090.253} C_VEL
LIN {X 0,Y 495.809,Z 486.725,A -85,B 0,C 180,E1 -6093.255,E2 -6093.255} C_VEL
LIN {X 0,Y 495.745,Z 486.732,A -85,B 0,C 180,E1 -6096.612,E2 -6096.612} C_VEL
LIN {X 0,Y 495.782,Z 486.728,A -85,B 0,C 180,E1 -6099.324,E2 -6099.324} C_VEL
LIN {X 0,Y 495.782,Z 486.729,A -85,B 0,C 180,E1 -6101.828,E2 -6101.828} C_VEL
LIN {X 0,Y 495.827,Z 486.724,A -85,B 0,C 180,E1 -6104.548,E2 -6104.548} C_VEL
LIN {X 0,Y 495.832,Z 486.723,A -85,B 0,C 180,E1 -6107.965,E2 -6107.965} C_VEL
LIN {X 0,Y 495.837,Z 486.722,A -85,B 0,C 180,E1 -6111.03,E2 -6111.03} C_VEL
LIN {X 0,Y 495.883,Z 486.715,A -85,B 0,C 180,E1 -6114.306,E2 -6114.306} C_VEL
LIN {X 0,Y 495.99,Z 486.702,A -85,B 0,C 180,E1 -6117.563,E2 -6117.563} C_VEL
LIN {X 0,Y 495.986,Z 486.704,A -85,B 0,C 180,E1 -6120.812,E2 -6120.812} C_VEL
LIN {X 0,Y 495.988,Z 486.704,A -85,B 0,C 180,E1 -6122.436,E2 -6122.436} C_VEL
LIN {X 0,Y 495.875,Z 486.718,A -85,B 0,C 180,E1 -6125.694,E2 -6125.694} C_VEL
LIN {X 0,Y 495.839,Z 486.722,A -85,B 0,C 180,E1 -6128.97,E2 -6128.97} C_VEL
LIN {X 0,Y 495.855,Z 486.719,A -85,B 0,C 180,E1 -6132.275,E2 -6132.275} C_VEL
LIN {X 0,Y 495.808,Z 486.726,A -85,B 0,C 180,E1 -6135.624,E2 -6135.624} C_VEL
LIN {X 0,Y 495.784,Z 486.731,A -85,B 0,C 180,E1 -6139.028,E2 -6139.028} C_VEL
LIN {X 0,Y 495.744,Z 486.734,A -85,B 0,C 180,E1 -6141.629,E2 -6141.629} C_VEL
LIN {X 0,Y 495.723,Z 486.735,A -85,B 0,C 180,E1 -6144.276,E2 -6144.276} C_VEL
LIN {X 0,Y 495.76,Z 486.732,A -85,B 0,C 180,E1 -6146.977,E2 -6146.977} C_VEL
LIN {X 0,Y 495.767,Z 486.73,A -85,B 0,C 180,E1 -6150.147,E2 -6150.147} C_VEL
LIN {X 0,Y 495.791,Z 486.727,A -85,B 0,C 180,E1 -6153.244,E2 -6153.244} C_VEL
LIN {X 0,Y 495.721,Z 486.736,A -85,B 0,C 180,E1 -6156.088,E2 -6156.088} C_VEL
LIN {X 0,Y 495.761,Z 486.733,A -85,B 0,C 180,E1 -6158.768,E2 -6158.768} C_VEL
LIN {X 0,Y 495.757,Z 486.733,A -85,B 0,C 180,E1 -6161.781,E2 -6161.781} C_VEL
LIN {X 0,Y 495.738,Z 486.731,A -85,B 0,C 180,E1 -6165.141,E2 -6165.141} C_VEL
LIN {X 0,Y 495.757,Z 486.728,A -85,B 0,C 180,E1 -6168.219,E2 -6168.219} C_VEL
LIN {X 0,Y 495.745,Z 486.743,A -85,B 0,C 180,E1 -6170.208,E2 -6170.208} C_VEL
LIN {X 0,Y 497.912,Z 497.609,A -85,B 0,C 180,E1 -6173.121,E2 -6173.121} C_VEL
LIN {X 0,Y 498.204,Z 501.768,A -85,B 0,C 180,E1 -6174.167,E2 -6174.167} C_VEL
LIN {X 0,Y 497.672,Z 514.934,A -85,B 0,C 180,E1 -6177.306,E2 -6177.306} C_VEL
LIN {X 0,Y 497.246,Z 528.12,A -85,B 0,C 180,E1 -6180.351,E2 -6180.351} C_VEL
LIN {X 0,Y 496.76,Z 543.374,A -85,B 0,C 180,E1 -6183.761,E2 -6183.761} C_VEL
LIN {X 0,Y 496.459,Z 556.688,A -85,B 0,C 180,E1 -6186.648,E2 -6186.648} C_VEL
LIN {X 0,Y 496.105,Z 571.953,A -85,B 0,C 180,E1 -6189.908,E2 -6189.908} C_VEL
LIN {X 0,Y 495.847,Z 586.213,A -85,B 0,C 180,E1 -6192.896,E2 -6192.896} C_VEL
LIN {X 0,Y 495.62,Z 598.529,A -85,B 0,C 180,E1 -6195.448,E2 -6195.448} C_VEL
LIN {X 0,Y 496.924,Z 610.13,A -85,B 0,C 180,E1 -6195.741,E2 -6195.741} C_VEL
LIN {X 0,Y 497.637,Z 616.616,A -85,B 0,C 180,E1 -6195.952,E2 -6195.952} C_VEL
LIN {X 0,Y 497.272,Z 629.659,A -85,B 0,C 180,E1 -6196.463,E2 -6196.463} C_VEL
LIN {X 0,Y 496.876,Z 641.85,A -85,B 0,C 180,E1 -6197.112,E2 -6197.112} C_VEL
LIN {X 0,Y 496.524,Z 653.887,A -85,B 0,C 180,E1 -6197.949,E2 -6197.949} C_VEL
LIN {X 0,Y 496.171,Z 664.503,A -85,B 0,C 180,E1 -6198.873,E2 -6198.873} C_VEL
LIN {X 0,Y 495.82,Z 673.198,A -85,B 0,C 180,E1 -6199.794,E2 -6199.794} C_VEL
LIN {X 0,Y 495.6,Z 681.248,A -85,B 0,C 180,E1 -6200.82,E2 -6200.82} C_VEL
LIN {X 0,Y 495.389,Z 689.131,A -85,B 0,C 180,E1 -6202.049,E2 -6202.049} C_VEL
LIN {X 0,Y 495.203,Z 696.393,A -85,B 0,C 180,E1 -6203.481,E2 -6203.481} C_VEL
LIN {X 0,Y 495.172,Z 701.243,A -85,B 0,C 180,E1 -6204.707,E2 -6204.707} C_VEL
LIN {X 0,Y 495.14,Z 704.949,A -85,B 0,C 180,E1 -6205.93,E2 -6205.93} C_VEL
LIN {X 0,Y 495.105,Z 706.854,A -85,B 0,C 180,E1 -6206.745,E2 -6206.745} C_VEL
LIN {X 0,Y 495.069,Z 708.285,A -85,B 0,C 180,E1 -6207.559,E2 -6207.559} C_VEL
LIN {X 0,Y 495.028,Z 709.3,A -85,B 0,C 180,E1 -6208.373,E2 -6208.373} C_VEL
LIN {X 0,Y 494.994,Z 709.916,A -85,B 0,C 180,E1 -6209.187,E2 -6209.187} C_VEL
LIN {X 0,Y 495.013,Z 710.13,A -85,B 0,C 180,E1 -6210,E2 -6210} C_VEL
LIN {X 0,Y 495.032,Z 709.271,A -85,B 0,C 180,E1 -6211.627,E2 -6211.627} C_VEL
LIN {X 0,Y 495.074,Z 708.242,A -85,B 0,C 180,E1 -6212.441,E2 -6212.441} C_VEL
LIN {X 0,Y 495.111,Z 706.79,A -85,B 0,C 180,E1 -6213.255,E2 -6213.255} C_VEL
LIN {X 0,Y 495.112,Z 703.743,A -85,B 0,C 180,E1 -6214.478,E2 -6214.478} C_VEL
LIN {X 0,Y 495.248,Z 698.437,A -85,B 0,C 180,E1 -6216.002,E2 -6216.002} C_VEL
LIN {X 0,Y 495.317,Z 692.274,A -85,B 0,C 180,E1 -6217.337,E2 -6217.337} C_VEL
LIN {X 0,Y 495.507,Z 685.15,A -85,B 0,C 180,E1 -6218.565,E2 -6218.565} C_VEL
LIN {X 0,Y 495.714,Z 676.245,A -85,B 0,C 180,E1 -6219.796,E2 -6219.796} C_VEL
LIN {X 0,Y 496.098,Z 666.156,A -85,B 0,C 180,E1 -6220.922,E2 -6220.922} C_VEL
LIN {X 0,Y 496.452,Z 655.984,A -85,B 0,C 180,E1 -6221.845,E2 -6221.845} C_VEL
LIN {X 0,Y 496.739,Z 644.532,A -85,B 0,C 180,E1 -6222.679,E2 -6222.679} C_VEL
LIN {X 0,Y 497.157,Z 632.156,A -85,B 0,C 180,E1 -6223.385,E2 -6223.385} C_VEL
LIN {X 0,Y 497.487,Z 620.305,A -85,B 0,C 180,E1 -6223.896,E2 -6223.896} C_VEL
LIN {X 0,Y 497.424,Z 613.745,A -85,B 0,C 180,E1 -6224.12,E2 -6224.12} C_VEL
LIN {X 0,Y 496.07,Z 603.37,A -85,B 0,C 180,E1 -6224.421,E2 -6224.421} C_VEL
LIN {X 0,Y 495.62,Z 597.703,A -85,B 0,C 180,E1 -6224.552,E2 -6224.552} C_VEL
LIN {X 0,Y 495.863,Z 581.974,A -85,B 0,C 180,E1 -6227.742,E2 -6227.742} C_VEL
LIN {X 0,Y 496.074,Z 567.086,A -85,B 0,C 180,E1 -6230.765,E2 -6230.765} C_VEL
LIN {X 0,Y 496.338,Z 551.375,A -85,B 0,C 180,E1 -6234.022,E2 -6234.022} C_VEL
LIN {X 0,Y 496.612,Z 535.585,A -85,B 0,C 180,E1 -6237.383,E2 -6237.383} C_VEL
LIN {X 0,Y 496.864,Z 521.994,A -85,B 0,C 180,E1 -6240.364,E2 -6240.364} C_VEL
LIN {X 0,Y 497.15,Z 509.498,A -85,B 0,C 180,E1 -6243.216,E2 -6243.216} C_VEL
LIN {X 0,Y 497.577,Z 497.27,A -85,B 0,C 180,E1 -6246.124,E2 -6246.124} C_VEL
LIN {X 0,Y 496.415,Z 490.024,A -85,B 0,C 180,E1 -6248.023,E2 -6248.023} C_VEL
LIN {X 0,Y 495.791,Z 486.731,A -85,B 0,C 180,E1 -6248.932,E2 -6248.932} C_VEL
LIN {X 0,Y 495.76,Z 486.733,A -85,B 0,C 180,E1 -6251.781,E2 -6251.781} C_VEL
LIN {X 0,Y 495.752,Z 486.737,A -85,B 0,C 180,E1 -6255.14,E2 -6255.14} C_VEL
LIN {X 0,Y 495.76,Z 486.734,A -85,B 0,C 180,E1 -6258.219,E2 -6258.219} C_VEL
LIN {X 0,Y 495.753,Z 486.733,A -85,B 0,C 180,E1 -6261.409,E2 -6261.409} C_VEL
LIN {X 0,Y 495.747,Z 486.733,A -85,B 0,C 180,E1 -6264.462,E2 -6264.462} C_VEL
LIN {X 0,Y 495.769,Z 486.732,A -85,B 0,C 180,E1 -6267.406,E2 -6267.406} C_VEL
LIN {X 0,Y 495.77,Z 486.729,A -85,B 0,C 180,E1 -6270.254,E2 -6270.254} C_VEL
LIN {X 0,Y 495.827,Z 486.722,A -85,B 0,C 180,E1 -6273.251,E2 -6273.251} C_VEL
LIN {X 0,Y 495.746,Z 486.732,A -85,B 0,C 180,E1 -6276.613,E2 -6276.613} C_VEL
LIN {X 0,Y 495.782,Z 486.726,A -85,B 0,C 180,E1 -6279.324,E2 -6279.324} C_VEL
LIN {X 0,Y 495.785,Z 486.727,A -85,B 0,C 180,E1 -6281.829,E2 -6281.829} C_VEL
LIN {X 0,Y 495.828,Z 486.724,A -85,B 0,C 180,E1 -6284.549,E2 -6284.549} C_VEL
LIN {X 0,Y 495.833,Z 486.722,A -85,B 0,C 180,E1 -6287.965,E2 -6287.965} C_VEL
LIN {X 0,Y 495.842,Z 486.723,A -85,B 0,C 180,E1 -6291.03,E2 -6291.03} C_VEL
LIN {X 0,Y 495.886,Z 486.719,A -85,B 0,C 180,E1 -6293.49,E2 -6293.49} C_VEL
LIN {X 0,Y 495.813,Z 486.725,A -85,B 0,C 180,E1 -6296.75,E2 -6296.75} C_VEL
LIN {X 0,Y 495.874,Z 486.719,A -85,B 0,C 180,E1 -6298.376,E2 -6298.376} C_VEL
LIN {X 0,Y 495.988,Z 486.705,A -85,B 0,C 180,E1 -6300.812,E2 -6300.812} C_VEL
LIN {X 0,Y 495.997,Z 486.704,A -85,B 0,C 180,E1 -6302.437,E2 -6302.437} C_VEL
LIN {X 0,Y 495.878,Z 486.718,A -85,B 0,C 180,E1 -6305.694,E2 -6305.694} C_VEL
LIN {X 0,Y 495.843,Z 486.72,A -85,B 0,C 180,E1 -6308.97,E2 -6308.97} C_VEL
LIN {X 0,Y 495.834,Z 486.724,A -85,B 0,C 180,E1 -6312.035,E2 -6312.035} C_VEL
LIN {X 0,Y 495.829,Z 486.724,A -85,B 0,C 180,E1 -6315.452,E2 -6315.452} C_VEL
LIN {X 0,Y 495.784,Z 486.735,A -85,B 0,C 180,E1 -6318.238,E2 -6318.238} C_VEL
LIN {X 0,Y 495.834,Z 486.726,A -85,B 0,C 180,E1 -6320.337,E2 -6320.337} C_VEL
LIN {X 0,Y 497.72,Z 494.457,A -85,B 0,C 180,E1 -6320.791,E2 -6320.791} C_VEL
LIN {X 0,Y 497.417,Z 505.096,A -85,B 0,C 180,E1 -6321.433,E2 -6321.433} C_VEL
LIN {X 0,Y 497.108,Z 515.476,A -85,B 0,C 180,E1 -6322.222,E2 -6322.222} C_VEL
LIN {X 0,Y 496.76,Z 525.13,A -85,B 0,C 180,E1 -6323.132,E2 -6323.132} C_VEL
LIN {X 0,Y 496.374,Z 534.653,A -85,B 0,C 180,E1 -6324.243,E2 -6324.243} C_VEL
LIN {X 0,Y 496.096,Z 542.504,A -85,B 0,C 180,E1 -6325.375,E2 -6325.375} C_VEL
LIN {X 0,Y 495.9,Z 548.348,A -85,B 0,C 180,E1 -6326.403,E2 -6326.403} C_VEL
LIN {X 0,Y 495.715,Z 553.221,A -85,B 0,C 180,E1 -6327.437,E2 -6327.437} C_VEL
LIN {X 0,Y 495.503,Z 558.45,A -85,B 0,C 180,E1 -6328.832,E2 -6328.832} C_VEL
LIN {X 0,Y 495.409,Z 561.912,A -85,B 0,C 180,E1 -6330.075,E2 -6330.075} C_VEL
LIN {X 0,Y 495.303,Z 564.887,A -85,B 0,C 180,E1 -6331.669,E2 -6331.669} C_VEL
LIN {X 0,Y 495.219,Z 566.257,A -85,B 0,C 180,E1 -6333.142,E2 -6333.142} C_VEL
LIN {X 0,Y 495.217,Z 566.353,A -85,B 0,C 180,E1 -6334.601,E2 -6334.601} C_VEL
LIN {X 0,Y 495.194,Z 565.291,A -85,B 0,C 180,E1 -6336.004,E2 -6336.004} C_VEL
LIN {X 0,Y 495.326,Z 563.095,A -85,B 0,C 180,E1 -6337.385,E2 -6337.385} C_VEL
LIN {X 0,Y 495.412,Z 559.838,A -85,B 0,C 180,E1 -6338.717,E2 -6338.717} C_VEL
LIN {X 0,Y 495.603,Z 554.249,A -85,B 0,C 180,E1 -6340.323,E2 -6340.323} C_VEL
LIN {X 0,Y 495.735,Z 549.06,A -85,B 0,C 180,E1 -6341.465,E2 -6341.465} C_VEL
LIN {X 0,Y 495.949,Z 543.116,A -85,B 0,C 180,E1 -6342.533,E2 -6342.533} C_VEL
LIN {X 0,Y 496.3,Z 534.689,A -85,B 0,C 180,E1 -6343.763,E2 -6343.763} C_VEL
LIN {X 0,Y 496.658,Z 525.157,A -85,B 0,C 180,E1 -6344.881,E2 -6344.881} C_VEL
LIN {X 0,Y 497.021,Z 514.826,A -85,B 0,C 180,E1 -6345.859,E2 -6345.859} C_VEL
LIN {X 0,Y 497.368,Z 503.66,A -85,B 0,C 180,E1 -6346.695,E2 -6346.695} C_VEL
LIN {X 0,Y 497.556,Z 493.38,A -85,B 0,C 180,E1 -6347.312,E2 -6347.312} C_VEL
LIN {X 0,Y 495.769,Z 486.733,A -85,B 0,C 180,E1 -6347.723,E2 -6347.723} C_VEL
LIN {X 0,Y 495.765,Z 486.732,A -85,B 0,C 180,E1 -6351.232,E2 -6351.232} C_VEL
LIN {X 0,Y 495.725,Z 486.736,A -85,B 0,C 180,E1 -6354.128,E2 -6354.128} C_VEL
LIN {X 0,Y 495.087,Z 486.814,A -85,B 0,C 180,E1 -6354.807,E2 -6354.807} C_VEL
LIN {X 0,Y 492.237,Z 487.169,A -85,B 0,C 180,E1 -6355.909,E2 -6355.909} C_VEL
LIN {X 0,Y 489.815,Z 487.472,A -85,B 0,C 180,E1 -6356.797,E2 -6356.797} C_VEL
LIN {X 0,Y 488.783,Z 487.6,A -85,B 0,C 180,E1 -6357.484,E2 -6357.484} C_VEL
LIN {X 0,Y 488.705,Z 487.609,A -85,B 0,C 180,E1 -6357.716,E2 -6357.716} C_VEL
LIN {X 0,Y 488.727,Z 487.606,A -85,B 0,C 180,E1 -6360.73,E2 -6360.73} C_VEL
LIN {X 0,Y 488.741,Z 487.606,A -85,B 0,C 180,E1 -6363.527,E2 -6363.527} C_VEL
LIN {X 0,Y 488.678,Z 487.613,A -85,B 0,C 180,E1 -6366.254,E2 -6366.254} C_VEL
LIN {X 0,Y 488.753,Z 487.606,A -85,B 0,C 180,E1 -6369.176,E2 -6369.176} C_VEL
LIN {X 0,Y 488.753,Z 487.606,A -85,B 0,C 180,E1 -6371.632,E2 -6371.632} C_VEL
LIN {X 0,Y 488.766,Z 487.606,A -85,B 0,C 180,E1 -6375,E2 -6375} C_VEL
LIN {X 0,Y 488.812,Z 487.596,A -85,B 0,C 180,E1 -6378.388,E2 -6378.388} C_VEL
LIN {X 0,Y 488.786,Z 487.6,A -85,B 0,C 180,E1 -6381.733,E2 -6381.733} C_VEL
LIN {X 0,Y 488.835,Z 487.594,A -85,B 0,C 180,E1 -6384.224,E2 -6384.224} C_VEL
LIN {X 0,Y 488.966,Z 487.577,A -85,B 0,C 180,E1 -6387.529,E2 -6387.529} C_VEL
LIN {X 0,Y 488.92,Z 487.583,A -85,B 0,C 180,E1 -6390.824,E2 -6390.824} C_VEL
LIN {X 0,Y 488.961,Z 487.578,A -85,B 0,C 180,E1 -6392.471,E2 -6392.471} C_VEL
LIN {X 0,Y 488.834,Z 487.596,A -85,B 0,C 180,E1 -6395.776,E2 -6395.776} C_VEL
LIN {X 0,Y 488.792,Z 487.598,A -85,B 0,C 180,E1 -6398.267,E2 -6398.267} C_VEL
LIN {X 0,Y 488.811,Z 487.6,A -85,B 0,C 180,E1 -6401.612,E2 -6401.612} C_VEL
LIN {X 0,Y 488.767,Z 487.605,A -85,B 0,C 180,E1 -6405,E2 -6405} C_VEL
LIN {X 0,Y 488.751,Z 487.603,A -85,B 0,C 180,E1 -6408.442,E2 -6408.442} C_VEL
LIN {X 0,Y 488.712,Z 487.611,A -85,B 0,C 180,E1 -6411.07,E2 -6411.07} C_VEL
LIN {X 0,Y 488.677,Z 487.615,A -85,B 0,C 180,E1 -6413.746,E2 -6413.746} C_VEL
LIN {X 0,Y 488.73,Z 487.61,A -85,B 0,C 180,E1 -6416.928,E2 -6416.928} C_VEL
LIN {X 0,Y 488.727,Z 487.607,A -85,B 0,C 180,E1 -6420.219,E2 -6420.219} C_VEL
LIN {X 0,Y 488.733,Z 487.606,A -85,B 0,C 180,E1 -6423.483,E2 -6423.483} C_VEL
LIN {X 0,Y 488.677,Z 487.613,A -85,B 0,C 180,E1 -6426.353,E2 -6426.353} C_VEL
LIN {X 0,Y 488.697,Z 487.611,A -85,B 0,C 180,E1 -6429.255,E2 -6429.255} C_VEL
LIN {X 0,Y 488.671,Z 487.613,A -85,B 0,C 180,E1 -6432.528,E2 -6432.528} C_VEL
LIN {X 0,Y 488.705,Z 487.61,A -85,B 0,C 180,E1 -6435.197,E2 -6435.197} C_VEL
LIN {X 0,Y 488.698,Z 487.61,A -85,B 0,C 180,E1 -6438.583,E2 -6438.583} C_VEL
LIN {X 0,Y 488.707,Z 487.612,A -85,B 0,C 180,E1 -6440.947,E2 -6440.947} C_VEL
LIN {X 0,Y 488.671,Z 487.615,A -85,B 0,C 180,E1 -6443.867,E2 -6443.867} C_VEL
LIN {X 0,Y 488.742,Z 487.608,A -85,B 0,C 180,E1 -6446.877,E2 -6446.877} C_VEL
LIN {X 0,Y 488.728,Z 487.608,A -85,B 0,C 180,E1 -6449.781,E2 -6449.781} C_VEL
LIN {X 0,Y 488.736,Z 487.608,A -85,B 0,C 180,E1 -6452.602,E2 -6452.602} C_VEL
LIN {X 0,Y 488.705,Z 487.612,A -85,B 0,C 180,E1 -6455.351,E2 -6455.351} C_VEL
LIN {X 0,Y 488.701,Z 487.609,A -85,B 0,C 180,E1 -6458.043,E2 -6458.043} C_VEL
LIN {X 0,Y 488.743,Z 487.606,A -85,B 0,C 180,E1 -6460.686,E2 -6460.686} C_VEL
LIN {X 0,Y 488.764,Z 487.601,A -85,B 0,C 180,E1 -6464.145,E2 -6464.145} C_VEL
LIN {X 0,Y 488.742,Z 487.607,A -85,B 0,C 180,E1 -6467.543,E2 -6467.543} C_VEL
LIN {X 0,Y 488.762,Z 487.601,A -85,B 0,C 180,E1 -6470.064,E2 -6470.064} C_VEL
LIN {X 0,Y 488.824,Z 487.595,A -85,B 0,C 180,E1 -6472.767,E2 -6472.767} C_VEL
LIN {X 0,Y 488.809,Z 487.601,A -85,B 0,C 180,E1 -6475.051,E2 -6475.051} C_VEL
LIN {X 0,Y 488.957,Z 487.578,A -85,B 0,C 180,E1 -6477.528,E2 -6477.528} C_VEL
LIN {X 0,Y 488.937,Z 487.582,A -85,B 0,C 180,E1 -6480.823,E2 -6480.823} C_VEL
LIN {X 0,Y 488.954,Z 487.58,A -85,B 0,C 180,E1 -6482.471,E2 -6482.471} C_VEL
LIN {X 0,Y 488.832,Z 487.595,A -85,B 0,C 180,E1 -6485.776,E2 -6485.776} C_VEL
LIN {X 0,Y 488.818,Z 487.595,A -85,B 0,C 180,E1 -6488.266,E2 -6488.266} C_VEL
LIN {X 0,Y 488.832,Z 487.595,A -85,B 0,C 180,E1 -6491.612,E2 -6491.612} C_VEL
LIN {X 0,Y 488.76,Z 487.604,A -85,B 0,C 180,E1 -6495,E2 -6495} C_VEL
LIN {X 0,Y 488.749,Z 487.604,A -85,B 0,C 180,E1 -6498.442,E2 -6498.442} C_VEL
LIN {X 0,Y 488.709,Z 487.609,A -85,B 0,C 180,E1 -6501.071,E2 -6501.071} C_VEL
LIN {X 0,Y 488.676,Z 487.614,A -85,B 0,C 180,E1 -6503.746,E2 -6503.746} C_VEL
LIN {X 0,Y 488.718,Z 487.61,A -85,B 0,C 180,E1 -6506.474,E2 -6506.474} C_VEL
LIN {X 0,Y 488.711,Z 487.612,A -85,B 0,C 180,E1 -6509.271,E2 -6509.271} C_VEL
LIN {X 0,Y 488.704,Z 487.609,A -85,B 0,C 180,E1 -6512.147,E2 -6512.147} C_VEL
LIN {X 0,Y 488.716,Z 487.61,A -85,B 0,C 180,E1 -6515.115,E2 -6515.115} C_VEL
LIN {X 0,Y 488.679,Z 487.613,A -85,B 0,C 180,E1 -6518.2,E2 -6518.2} C_VEL
LIN {X 0,Y 488.72,Z 487.61,A -85,B 0,C 180,E1 -6520.345,E2 -6520.345} C_VEL
LIN {X 0,Y 488.686,Z 487.611,A -85,B 0,C 180,E1 -6523.655,E2 -6523.655} C_VEL
LIN {X 0,Y 488.679,Z 487.611,A -85,B 0,C 180,E1 -6526.345,E2 -6526.345} C_VEL
LIN {X 0,Y 488.735,Z 487.604,A -85,B 0,C 180,E1 -6529.677,E2 -6529.677} C_VEL
LIN {X 0,Y 488.739,Z 487.699,A -85,B 0,C 180,E1 -6529.947,E2 -6529.947} C_VEL
LIN {X 0,Y 490.972,Z 499.063,A -85,B 0,C 180,E1 -6533.043,E2 -6533.043} C_VEL
LIN {X 0,Y 491.282,Z 503.167,A -85,B 0,C 180,E1 -6534.089,E2 -6534.089} C_VEL
LIN {X 0,Y 490.725,Z 515.282,A -85,B 0,C 180,E1 -6537.028,E2 -6537.028} C_VEL
LIN {X 0,Y 490.273,Z 528.465,A -85,B 0,C 180,E1 -6540.123,E2 -6540.123} C_VEL
LIN {X 0,Y 489.823,Z 541.949,A -85,B 0,C 180,E1 -6543.2,E2 -6543.2} C_VEL
LIN {X 0,Y 489.447,Z 555.863,A -85,B 0,C 180,E1 -6546.293,E2 -6546.293} C_VEL
LIN {X 0,Y 489.05,Z 572.173,A -85,B 0,C 180,E1 -6549.824,E2 -6549.824} C_VEL
LIN {X 0,Y 488.732,Z 587.337,A -85,B 0,C 180,E1 -6553.07,E2 -6553.07} C_VEL
LIN {X 0,Y 488.563,Z 597.573,A -85,B 0,C 180,E1 -6555.233,E2 -6555.233} C_VEL
LIN {X 0,Y 489.949,Z 610.752,A -85,B 0,C 180,E1 -6555.581,E2 -6555.581} C_VEL
LIN {X 0,Y 490.66,Z 617.099,A -85,B 0,C 180,E1 -6555.801,E2 -6555.801} C_VEL
LIN {X 0,Y 490.298,Z 629.745,A -85,B 0,C 180,E1 -6556.319,E2 -6556.319} C_VEL
LIN {X 0,Y 489.876,Z 641.406,A -85,B 0,C 180,E1 -6556.962,E2 -6556.962} C_VEL
LIN {X 0,Y 489.51,Z 652.864,A -85,B 0,C 180,E1 -6557.774,E2 -6557.774} C_VEL
LIN {X 0,Y 489.118,Z 663.479,A -85,B 0,C 180,E1 -6558.71,E2 -6558.71} C_VEL
LIN {X 0,Y 488.787,Z 672.183,A -85,B 0,C 180,E1 -6559.646,E2 -6559.646} C_VEL
LIN {X 0,Y 488.531,Z 680.233,A -85,B 0,C 180,E1 -6560.686,E2 -6560.686} C_VEL
LIN {X 0,Y 488.338,Z 688.125,A -85,B 0,C 180,E1 -6561.934,E2 -6561.934} C_VEL
LIN {X 0,Y 488.141,Z 695.387,A -85,B 0,C 180,E1 -6563.386,E2 -6563.386} C_VEL
LIN {X 0,Y 488.111,Z 700.238,A -85,B 0,C 180,E1 -6564.63,E2 -6564.63} C_VEL
LIN {X 0,Y 488.077,Z 703.943,A -85,B 0,C 180,E1 -6565.871,E2 -6565.871} C_VEL
LIN {X 0,Y 488.058,Z 705.85,A -85,B 0,C 180,E1 -6566.698,E2 -6566.698} C_VEL
LIN {X 0,Y 488.029,Z 707.28,A -85,B 0,C 180,E1 -6567.524,E2 -6567.524} C_VEL
LIN {X 0,Y 487.995,Z 708.294,A -85,B 0,C 180,E1 -6568.35,E2 -6568.35} C_VEL
LIN {X 0,Y 488.007,Z 709.118,A -85,B 0,C 180,E1 -6570,E2 -6570} C_VEL
LIN {X 0,Y 488.002,Z 708.245,A -85,B 0,C 180,E1 -6571.651,E2 -6571.651} C_VEL
LIN {X 0,Y 488.038,Z 707.205,A -85,B 0,C 180,E1 -6572.476,E2 -6572.476} C_VEL
LIN {X 0,Y 488.07,Z 705.745,A -85,B 0,C 180,E1 -6573.302,E2 -6573.302} C_VEL
LIN {X 0,Y 488.064,Z 702.684,A -85,B 0,C 180,E1 -6574.543,E2 -6574.543} C_VEL
LIN {X 0,Y 488.189,Z 697.53,A -85,B 0,C 180,E1 -6576.046,E2 -6576.046} C_VEL
LIN {X 0,Y 488.255,Z 691.172,A -85,B 0,C 180,E1 -6577.444,E2 -6577.444} C_VEL
LIN {X 0,Y 488.452,Z 684.029,A -85,B 0,C 180,E1 -6578.69,E2 -6578.69} C_VEL
LIN {X 0,Y 488.662,Z 675.101,A -85,B 0,C 180,E1 -6579.938,E2 -6579.938} C_VEL
LIN {X 0,Y 489.082,Z 664.991,A -85,B 0,C 180,E1 -6581.081,E2 -6581.081} C_VEL
LIN {X 0,Y 489.428,Z 654.793,A -85,B 0,C 180,E1 -6582.018,E2 -6582.018} C_VEL
LIN {X 0,Y 489.73,Z 644.14,A -85,B 0,C 180,E1 -6582.81,E2 -6582.81} C_VEL
LIN {X 0,Y 490.133,Z 631.925,A -85,B 0,C 180,E1 -6583.527,E2 -6583.527} C_VEL
LIN {X 0,Y 490.546,Z 619.055,A -85,B 0,C 180,E1 -6584.097,E2 -6584.097} C_VEL
LIN {X 0,Y 490.456,Z 614.501,A -85,B 0,C 180,E1 -6584.258,E2 -6584.258} C_VEL
LIN {X 0,Y 489.159,Z 604.341,A -85,B 0,C 180,E1 -6584.576,E2 -6584.576} C_VEL
LIN {X 0,Y 488.564,Z 596.525,A -85,B 0,C 180,E1 -6584.767,E2 -6584.767} C_VEL
LIN {X 0,Y 488.798,Z 580.903,A -85,B 0,C 180,E1 -6587.981,E2 -6587.981} C_VEL
LIN {X 0,Y 489.012,Z 565.049,A -85,B 0,C 180,E1 -6591.278,E2 -6591.278} C_VEL
LIN {X 0,Y 489.334,Z 549.29,A -85,B 0,C 180,E1 -6594.615,E2 -6594.615} C_VEL
LIN {X 0,Y 489.612,Z 534.606,A -85,B 0,C 180,E1 -6597.808,E2 -6597.808} C_VEL
LIN {X 0,Y 489.962,Z 520.015,A -85,B 0,C 180,E1 -6601.09,E2 -6601.09} C_VEL
LIN {X 0,Y 490.328,Z 506.635,A -85,B 0,C 180,E1 -6604.235,E2 -6604.235} C_VEL
LIN {X 0,Y 490.63,Z 498.216,A -85,B 0,C 180,E1 -6606.297,E2 -6606.297} C_VEL
LIN {X 0,Y 489.148,Z 489.704,A -85,B 0,C 180,E1 -6608.596,E2 -6608.596} C_VEL
LIN {X 0,Y 488.745,Z 487.607,A -85,B 0,C 180,E1 -6609.25,E2 -6609.25} C_VEL
LIN {X 0,Y 488.695,Z 487.615,A -85,B 0,C 180,E1 -6612.526,E2 -6612.526} C_VEL
LIN {X 0,Y 488.715,Z 487.613,A -85,B 0,C 180,E1 -6615.199,E2 -6615.199} C_VEL
LIN {X 0,Y 488.711,Z 487.613,A -85,B 0,C 180,E1 -6618.4,E2 -6618.4} C_VEL
LIN {X 0,Y 488.707,Z 487.613,A -85,B 0,C 180,E1 -6620.948,E2 -6620.948} C_VEL
LIN {X 0,Y 488.673,Z 487.616,A -85,B 0,C 180,E1 -6623.868,E2 -6623.868} C_VEL
LIN {X 0,Y 488.738,Z 487.606,A -85,B 0,C 180,E1 -6626.877,E2 -6626.877} C_VEL
LIN {X 0,Y 488.727,Z 487.61,A -85,B 0,C 180,E1 -6629.781,E2 -6629.781} C_VEL
LIN {X 0,Y 488.795,Z 487.597,A -85,B 0,C 180,E1 -6633.057,E2 -6633.057} C_VEL
LIN {X 0,Y 488.683,Z 487.612,A -85,B 0,C 180,E1 -6636.254,E2 -6636.254} C_VEL
LIN {X 0,Y 488.75,Z 487.602,A -85,B 0,C 180,E1 -6639.176,E2 -6639.176} C_VEL
LIN {X 0,Y 488.753,Z 487.603,A -85,B 0,C 180,E1 -6641.632,E2 -6641.632} C_VEL
LIN {X 0,Y 488.765,Z 487.601,A -85,B 0,C 180,E1 -6645,E2 -6645} C_VEL
LIN {X 0,Y 488.81,Z 487.597,A -85,B 0,C 180,E1 -6648.388,E2 -6648.388} C_VEL
LIN {X 0,Y 488.82,Z 487.594,A -85,B 0,C 180,E1 -6651.734,E2 -6651.734} C_VEL
LIN {X 0,Y 488.859,Z 487.591,A -85,B 0,C 180,E1 -6654.224,E2 -6654.224} C_VEL
LIN {X 0,Y 488.957,Z 487.579,A -85,B 0,C 180,E1 -6657.529,E2 -6657.529} C_VEL
LIN {X 0,Y 488.939,Z 487.583,A -85,B 0,C 180,E1 -6660.824,E2 -6660.824} C_VEL
LIN {X 0,Y 488.965,Z 487.58,A -85,B 0,C 180,E1 -6662.472,E2 -6662.472} C_VEL
LIN {X 0,Y 488.836,Z 487.595,A -85,B 0,C 180,E1 -6665.776,E2 -6665.776} C_VEL
LIN {X 0,Y 488.821,Z 487.598,A -85,B 0,C 180,E1 -6668.267,E2 -6668.267} C_VEL
LIN {X 0,Y 488.811,Z 487.597,A -85,B 0,C 180,E1 -6671.613,E2 -6671.613} C_VEL
LIN {X 0,Y 488.767,Z 487.605,A -85,B 0,C 180,E1 -6675.001,E2 -6675.001} C_VEL
LIN {X 0,Y 488.752,Z 487.611,A -85,B 0,C 180,E1 -6678.443,E2 -6678.443} C_VEL
LIN {X 0,Y 488.785,Z 487.703,A -85,B 0,C 180,E1 -6680.132,E2 -6680.132} C_VEL
LIN {X 0,Y 490.857,Z 496.029,A -85,B 0,C 180,E1 -6680.631,E2 -6680.631} C_VEL
LIN {X 0,Y 490.562,Z 507.837,A -85,B 0,C 180,E1 -6681.373,E2 -6681.373} C_VEL
LIN {X 0,Y 490.164,Z 518.381,A -85,B 0,C 180,E1 -6682.221,E2 -6682.221} C_VEL
LIN {X 0,Y 489.743,Z 529.153,A -85,B 0,C 180,E1 -6683.302,E2 -6683.302} C_VEL
LIN {X 0,Y 489.397,Z 537.795,A -85,B 0,C 180,E1 -6684.385,E2 -6684.385} C_VEL
LIN {X 0,Y 489.09,Z 545.265,A -85,B 0,C 180,E1 -6685.537,E2 -6685.537} C_VEL
LIN {X 0,Y 488.823,Z 552.578,A -85,B 0,C 180,E1 -6686.95,E2 -6686.95} C_VEL
LIN {X 0,Y 488.561,Z 558.124,A -85,B 0,C 180,E1 -6688.341,E2 -6688.341} C_VEL
LIN {X 0,Y 488.443,Z 562.327,A -85,B 0,C 180,E1 -6689.763,E2 -6689.763} C_VEL
LIN {X 0,Y 488.329,Z 565.279,A -85,B 0,C 180,E1 -6691.206,E2 -6691.206} C_VEL
LIN {X 0,Y 488.253,Z 566.573,A -85,B 0,C 180,E1 -6692.181,E2 -6692.181} C_VEL
LIN {X 0,Y 488.22,Z 567.397,A -85,B 0,C 180,E1 -6693.392,E2 -6693.392} C_VEL
LIN {X 0,Y 488.209,Z 567.288,A -85,B 0,C 180,E1 -6694.86,E2 -6694.86} C_VEL
LIN {X 0,Y 488.211,Z 566.003,A -85,B 0,C 180,E1 -6696.279,E2 -6696.279} C_VEL
LIN {X 0,Y 488.327,Z 563.596,A -85,B 0,C 180,E1 -6697.668,E2 -6697.668} C_VEL
LIN {X 0,Y 488.428,Z 560.139,A -85,B 0,C 180,E1 -6699.012,E2 -6699.012} C_VEL
LIN {X 0,Y 488.598,Z 555.524,A -85,B 0,C 180,E1 -6700.337,E2 -6700.337} C_VEL
LIN {X 0,Y 488.763,Z 549.849,A -85,B 0,C 180,E1 -6701.607,E2 -6701.607} C_VEL
LIN {X 0,Y 489.073,Z 542.721,A -85,B 0,C 180,E1 -6702.872,E2 -6702.872} C_VEL
LIN {X 0,Y 489.45,Z 533.972,A -85,B 0,C 180,E1 -6704.114,E2 -6704.114} C_VEL
LIN {X 0,Y 489.806,Z 524.738,A -85,B 0,C 180,E1 -6705.178,E2 -6705.178} C_VEL
LIN {X 0,Y 490.152,Z 515.132,A -85,B 0,C 180,E1 -6706.075,E2 -6706.075} C_VEL
LIN {X 0,Y 490.466,Z 505.4,A -85,B 0,C 180,E1 -6706.818,E2 -6706.818} C_VEL
LIN {X 0,Y 490.777,Z 495.247,A -85,B 0,C 180,E1 -6707.444,E2 -6707.444} C_VEL
LIN {X 0,Y 488.729,Z 487.61,A -85,B 0,C 180,E1 -6707.916,E2 -6707.916} C_VEL
LIN {X 0,Y 488.705,Z 487.613,A -85,B 0,C 180,E1 -6710.948,E2 -6710.948} C_VEL
LIN {X 0,Y 488.672,Z 487.614,A -85,B 0,C 180,E1 -6714.129,E2 -6714.129} C_VEL
LIN {X 0,Y 488.744,Z 487.607,A -85,B 0,C 180,E1 -6716.877,E2 -6716.877} C_VEL
LIN {X 0,Y 488.705,Z 487.609,A -85,B 0,C 180,E1 -6717.716,E2 -6717.716} C_VEL
LIN {X 0,Y 488.06,Z 487.693,A -85,B 0,C 180,E1 -6718.404,E2 -6718.404} C_VEL
LIN {X 0,Y 485.24,Z 488.049,A -85,B 0,C 180,E1 -6719.521,E2 -6719.521} C_VEL
LIN {X 0,Y 482.835,Z 488.347,A -85,B 0,C 180,E1 -6720.421,E2 -6720.421} C_VEL
LIN {X 0,Y 481.787,Z 488.474,A -85,B 0,C 180,E1 -6721.116,E2 -6721.116} C_VEL
LIN {X 0,Y 481.695,Z 488.483,A -85,B 0,C 180,E1 -6721.352,E2 -6721.352} C_VEL
LIN {X 0,Y 481.68,Z 488.486,A -85,B 0,C 180,E1 -6724.041,E2 -6724.041} C_VEL
LIN {X 0,Y 481.68,Z 488.484,A -85,B 0,C 180,E1 -6726.812,E2 -6726.812} C_VEL
LIN {X 0,Y 481.701,Z 488.483,A -85,B 0,C 180,E1 -6729.503,E2 -6729.503} C_VEL
LIN {X 0,Y 481.694,Z 488.483,A -85,B 0,C 180,E1 -6732.158,E2 -6732.158} C_VEL
LIN {X 0,Y 481.748,Z 488.477,A -85,B 0,C 180,E1 -6734.776,E2 -6734.776} C_VEL
LIN {X 0,Y 481.757,Z 488.475,A -85,B 0,C 180,E1 -6738.215,E2 -6738.215} C_VEL
LIN {X 0,Y 481.742,Z 488.477,A -85,B 0,C 180,E1 -6741.611,E2 -6741.611} C_VEL
LIN {X 0,Y 481.794,Z 488.471,A -85,B 0,C 180,E1 -6744.139,E2 -6744.139} C_VEL
LIN {X 0,Y 481.933,Z 488.454,A -85,B 0,C 180,E1 -6747.492,E2 -6747.492} C_VEL
LIN {X 0,Y 481.943,Z 488.453,A -85,B 0,C 180,E1 -6750,E2 -6750} C_VEL
LIN {X 0,Y 481.927,Z 488.454,A -85,B 0,C 180,E1 -6752.507,E2 -6752.507} C_VEL
LIN {X 0,Y 481.793,Z 488.472,A -85,B 0,C 180,E1 -6755.861,E2 -6755.861} C_VEL
LIN {X 0,Y 481.746,Z 488.476,A -85,B 0,C 180,E1 -6758.389,E2 -6758.389} C_VEL
LIN {X 0,Y 481.756,Z 488.477,A -85,B 0,C 180,E1 -6761.785,E2 -6761.785} C_VEL
LIN {X 0,Y 481.748,Z 488.477,A -85,B 0,C 180,E1 -6765.224,E2 -6765.224} C_VEL
LIN {X 0,Y 481.712,Z 488.48,A -85,B 0,C 180,E1 -6768.722,E2 -6768.722} C_VEL
LIN {X 0,Y 481.651,Z 488.489,A -85,B 0,C 180,E1 -6771.394,E2 -6771.394} C_VEL
LIN {X 0,Y 481.655,Z 488.488,A -85,B 0,C 180,E1 -6774.114,E2 -6774.114} C_VEL
LIN {X 0,Y 481.699,Z 488.484,A -85,B 0,C 180,E1 -6777.127,E2 -6777.127} C_VEL
LIN {X 0,Y 481.677,Z 488.487,A -85,B 0,C 180,E1 -6779.741,E2 -6779.741} C_VEL
LIN {X 0,Y 481.675,Z 488.487,A -85,B 0,C 180,E1 -6782.674,E2 -6782.674} C_VEL
LIN {X 0,Y 481.635,Z 488.492,A -85,B 0,C 180,E1 -6785.71,E2 -6785.71} C_VEL
LIN {X 0,Y 481.67,Z 488.49,A -85,B 0,C 180,E1 -6788.859,E2 -6788.859} C_VEL
LIN {X 0,Y 481.633,Z 488.491,A -85,B 0,C 180,E1 -6792.162,E2 -6792.162} C_VEL
LIN {X 0,Y 481.657,Z 488.488,A -85,B 0,C 180,E1 -6795.542,E2 -6795.542} C_VEL
LIN {X 0,Y 481.652,Z 488.49,A -85,B 0,C 180,E1 -6798.957,E2 -6798.957} C_VEL
LIN {X 0,Y 481.652,Z 488.49,A -85,B 0,C 180,E1 -6801.993,E2 -6801.993} C_VEL
LIN {X 0,Y 481.691,Z 488.485,A -85,B 0,C 180,E1 -6805.318,E2 -6805.318} C_VEL
LIN {X 0,Y 481.649,Z 488.49,A -85,B 0,C 180,E1 -6808.311,E2 -6808.311} C_VEL
LIN {X 0,Y 481.704,Z 488.485,A -85,B 0,C 180,E1 -6811.218,E2 -6811.218} C_VEL
LIN {X 0,Y 481.677,Z 488.486,A -85,B 0,C 180,E1 -6814.041,E2 -6814.041} C_VEL
LIN {X 0,Y 481.677,Z 488.486,A -85,B 0,C 180,E1 -6816.812,E2 -6816.812} C_VEL
LIN {X 0,Y 481.698,Z 488.483,A -85,B 0,C 180,E1 -6819.502,E2 -6819.502} C_VEL
LIN {X 0,Y 481.692,Z 488.483,A -85,B 0,C 180,E1 -6822.158,E2 -6822.158} C_VEL
LIN {X 0,Y 481.745,Z 488.48,A -85,B 0,C 180,E1 -6824.776,E2 -6824.776} C_VEL
LIN {X 0,Y 481.754,Z 488.475,A -85,B 0,C 180,E1 -6828.215,E2 -6828.215} C_VEL
LIN {X 0,Y 481.739,Z 488.478,A -85,B 0,C 180,E1 -6831.611,E2 -6831.611} C_VEL
LIN {X 0,Y 481.798,Z 488.47,A -85,B 0,C 180,E1 -6834.139,E2 -6834.139} C_VEL
LIN {X 0,Y 481.924,Z 488.455,A -85,B 0,C 180,E1 -6837.492,E2 -6837.492} C_VEL
LIN {X 0,Y 481.889,Z 488.461,A -85,B 0,C 180,E1 -6840.835,E2 -6840.835} C_VEL
LIN {X 0,Y 481.92,Z 488.457,A -85,B 0,C 180,E1 -6842.507,E2 -6842.507} C_VEL
LIN {X 0,Y 481.792,Z 488.472,A -85,B 0,C 180,E1 -6845.861,E2 -6845.861} C_VEL
LIN {X 0,Y 481.763,Z 488.475,A -85,B 0,C 180,E1 -6848.388,E2 -6848.388} C_VEL
LIN {X 0,Y 481.797,Z 488.471,A -85,B 0,C 180,E1 -6851.784,E2 -6851.784} C_VEL
LIN {X 0,Y 481.742,Z 488.477,A -85,B 0,C 180,E1 -6855.224,E2 -6855.224} C_VEL
LIN {X 0,Y 481.711,Z 488.482,A -85,B 0,C 180,E1 -6858.722,E2 -6858.722} C_VEL
LIN {X 0,Y 481.647,Z 488.489,A -85,B 0,C 180,E1 -6861.395,E2 -6861.395} C_VEL
LIN {X 0,Y 481.658,Z 488.487,A -85,B 0,C 180,E1 -6864.114,E2 -6864.114} C_VEL
LIN {X 0,Y 481.695,Z 488.483,A -85,B 0,C 180,E1 -6867.126,E2 -6867.126} C_VEL
LIN {X 0,Y 481.675,Z 488.486,A -85,B 0,C 180,E1 -6869.741,E2 -6869.741} C_VEL
LIN {X 0,Y 481.672,Z 488.489,A -85,B 0,C 180,E1 -6872.674,E2 -6872.674} C_VEL
LIN {X 0,Y 481.637,Z 488.491,A -85,B 0,C 180,E1 -6875.709,E2 -6875.709} C_VEL
LIN {X 0,Y 481.67,Z 488.487,A -85,B 0,C 180,E1 -6878.859,E2 -6878.859} C_VEL
LIN {X 0,Y 481.654,Z 488.489,A -85,B 0,C 180,E1 -6881.913,E2 -6881.913} C_VEL
LIN {X 0,Y 481.656,Z 488.489,A -85,B 0,C 180,E1 -6884.458,E2 -6884.458} C_VEL
LIN {X 0,Y 481.647,Z 488.487,A -85,B 0,C 180,E1 -6887.839,E2 -6887.839} C_VEL
LIN {X 0,Y 481.723,Z 488.621,A -85,B 0,C 180,E1 -6889.673,E2 -6889.673} C_VEL
LIN {X 0,Y 484.064,Z 500.598,A -85,B 0,C 180,E1 -6892.99,E2 -6892.99} C_VEL
LIN {X 0,Y 484.371,Z 504.393,A -85,B 0,C 180,E1 -6893.978,E2 -6893.978} C_VEL
LIN {X 0,Y 483.753,Z 516.635,A -85,B 0,C 180,E1 -6896.989,E2 -6896.989} C_VEL
LIN {X 0,Y 483.273,Z 529.792,A -85,B 0,C 180,E1 -6900.127,E2 -6900.127} C_VEL
LIN {X 0,Y 482.727,Z 544.957,A -85,B 0,C 180,E1 -6903.638,E2 -6903.638} C_VEL
LIN {X 0,Y 482.336,Z 558.197,A -85,B 0,C 180,E1 -6906.63,E2 -6906.63} C_VEL
LIN {X 0,Y 481.958,Z 573.342,A -85,B 0,C 180,E1 -6909.96,E2 -6909.96} C_VEL
LIN {X 0,Y 481.639,Z 588.464,A -85,B 0,C 180,E1 -6913.25,E2 -6913.25} C_VEL
LIN {X 0,Y 481.472,Z 596.612,A -85,B 0,C 180,E1 -6915.011,E2 -6915.011} C_VEL
LIN {X 0,Y 482.983,Z 611.492,A -85,B 0,C 180,E1 -6915.422,E2 -6915.422} C_VEL
LIN {X 0,Y 483.708,Z 617.557,A -85,B 0,C 180,E1 -6915.646,E2 -6915.646} C_VEL
LIN {X 0,Y 483.337,Z 629.796,A -85,B 0,C 180,E1 -6916.172,E2 -6916.172} C_VEL
LIN {X 0,Y 482.825,Z 642.136,A -85,B 0,C 180,E1 -6916.886,E2 -6916.886} C_VEL
LIN {X 0,Y 482.455,Z 652.836,A -85,B 0,C 180,E1 -6917.674,E2 -6917.674} C_VEL
LIN {X 0,Y 482.043,Z 663.532,A -85,B 0,C 180,E1 -6918.649,E2 -6918.649} C_VEL
LIN {X 0,Y 481.671,Z 672.896,A -85,B 0,C 180,E1 -6919.704,E2 -6919.704} C_VEL
LIN {X 0,Y 481.396,Z 682.03,A -85,B 0,C 180,E1 -6920.971,E2 -6920.971} C_VEL
LIN {X 0,Y 481.207,Z 689.399,A -85,B 0,C 180,E1 -6922.236,E2 -6922.236} C_VEL
LIN {X 0,Y 481.087,Z 696.033,A -85,B 0,C 180,E1 -6923.685,E2 -6923.685} C_VEL
LIN {X 0,Y 481.024,Z 700.584,A -85,B 0,C 180,E1 -6924.971,E2 -6924.971} C_VEL
LIN {X 0,Y 481.018,Z 702.938,A -85,B 0,C 180,E1 -6925.811,E2 -6925.811} C_VEL
LIN {X 0,Y 481.013,Z 704.845,A -85,B 0,C 180,E1 -6926.65,E2 -6926.65} C_VEL
LIN {X 0,Y 480.989,Z 706.275,A -85,B 0,C 180,E1 -6927.488,E2 -6927.488} C_VEL
LIN {X 0,Y 480.961,Z 707.288,A -85,B 0,C 180,E1 -6928.325,E2 -6928.325} C_VEL
LIN {X 0,Y 481,Z 708.106,A -85,B 0,C 180,E1 -6930,E2 -6930} C_VEL
LIN {X 0,Y 480.97,Z 707.22,A -85,B 0,C 180,E1 -6931.675,E2 -6931.675} C_VEL
LIN {X 0,Y 481.002,Z 706.169,A -85,B 0,C 180,E1 -6932.512,E2 -6932.512} C_VEL
LIN {X 0,Y 481.028,Z 704.701,A -85,B 0,C 180,E1 -6933.35,E2 -6933.35} C_VEL
LIN {X 0,Y 481.021,Z 701.626,A -85,B 0,C 180,E1 -6934.609,E2 -6934.609} C_VEL
LIN {X 0,Y 481.109,Z 697.486,A -85,B 0,C 180,E1 -6935.869,E2 -6935.869} C_VEL
LIN {X 0,Y 481.177,Z 691.123,A -85,B 0,C 180,E1 -6937.343,E2 -6937.343} C_VEL
LIN {X 0,Y 481.358,Z 684.192,A -85,B 0,C 180,E1 -6938.607,E2 -6938.607} C_VEL
LIN {X 0,Y 481.549,Z 675.601,A -85,B 0,C 180,E1 -6939.874,E2 -6939.874} C_VEL
LIN {X 0,Y 481.966,Z 665.83,A -85,B 0,C 180,E1 -6941.034,E2 -6941.034} C_VEL
LIN {X 0,Y 482.333,Z 656.248,A -85,B 0,C 180,E1 -6941.964,E2 -6941.964} C_VEL
LIN {X 0,Y 482.628,Z 645.351,A -85,B 0,C 180,E1 -6942.831,E2 -6942.831} C_VEL
LIN {X 0,Y 483.101,Z 633.701,A -85,B 0,C 180,E1 -6943.567,E2 -6943.567} C_VEL
LIN {X 0,Y 483.548,Z 620.42,A -85,B 0,C 180,E1 -6944.198,E2 -6944.198} C_VEL
LIN {X 0,Y 483.388,Z 614.744,A -85,B 0,C 180,E1 -6944.417,E2 -6944.417} C_VEL
LIN {X 0,Y 482.289,Z 605.88,A -85,B 0,C 180,E1 -6944.721,E2 -6944.721} C_VEL
LIN {X 0,Y 481.487,Z 595.342,A -85,B 0,C 180,E1 -6944.989,E2 -6944.989} C_VEL
LIN {X 0,Y 481.72,Z 580.161,A -85,B 0,C 180,E1 -6948.17,E2 -6948.17} C_VEL
LIN {X 0,Y 481.943,Z 565.01,A -85,B 0,C 180,E1 -6951.381,E2 -6951.381} C_VEL
LIN {X 0,Y 482.278,Z 549.304,A -85,B 0,C 180,E1 -6954.769,E2 -6954.769} C_VEL
LIN {X 0,Y 482.565,Z 535.73,A -85,B 0,C 180,E1 -6957.778,E2 -6957.778} C_VEL
LIN {X 0,Y 482.892,Z 522.387,A -85,B 0,C 180,E1 -6960.831,E2 -6960.831} C_VEL
LIN {X 0,Y 483.214,Z 510.927,A -85,B 0,C 180,E1 -6963.552,E2 -6963.552} C_VEL
LIN {X 0,Y 483.709,Z 499.821,A -85,B 0,C 180,E1 -6966.305,E2 -6966.305} C_VEL
LIN {X 0,Y 482.406,Z 492.089,A -85,B 0,C 180,E1 -6968.423,E2 -6968.423} C_VEL
LIN {X 0,Y 481.692,Z 488.484,A -85,B 0,C 180,E1 -6969.487,E2 -6969.487} C_VEL
LIN {X 0,Y 481.651,Z 488.492,A -85,B 0,C 180,E1 -6972.161,E2 -6972.161} C_VEL
LIN {X 0,Y 481.663,Z 488.491,A -85,B 0,C 180,E1 -6975.543,E2 -6975.543} C_VEL
LIN {X 0,Y 481.66,Z 488.491,A -85,B 0,C 180,E1 -6978.959,E2 -6978.959} C_VEL
LIN {X 0,Y 481.654,Z 488.488,A -85,B 0,C 180,E1 -6981.994,E2 -6981.994} C_VEL
LIN {X 0,Y 481.687,Z 488.484,A -85,B 0,C 180,E1 -6985.318,E2 -6985.318} C_VEL
LIN {X 0,Y 481.648,Z 488.488,A -85,B 0,C 180,E1 -6988.312,E2 -6988.312} C_VEL
LIN {X 0,Y 481.703,Z 488.483,A -85,B 0,C 180,E1 -6991.219,E2 -6991.219} C_VEL
LIN {X 0,Y 481.692,Z 488.483,A -85,B 0,C 180,E1 -6994.042,E2 -6994.042} C_VEL
LIN {X 0,Y 481.678,Z 488.484,A -85,B 0,C 180,E1 -6996.812,E2 -6996.812} C_VEL
LIN {X 0,Y 481.699,Z 488.481,A -85,B 0,C 180,E1 -6999.503,E2 -6999.503} C_VEL
LIN {X 0,Y 481.696,Z 488.483,A -85,B 0,C 180,E1 -7002.158,E2 -7002.158} C_VEL
LIN {X 0,Y 481.746,Z 488.477,A -85,B 0,C 180,E1 -7004.776,E2 -7004.776} C_VEL
LIN {X 0,Y 481.755,Z 488.476,A -85,B 0,C 180,E1 -7008.215,E2 -7008.215} C_VEL
LIN {X 0,Y 481.766,Z 488.472,A -85,B 0,C 180,E1 -7011.612,E2 -7011.612} C_VEL
LIN {X 0,Y 481.82,Z 488.468,A -85,B 0,C 180,E1 -7014.14,E2 -7014.14} C_VEL
LIN {X 0,Y 481.922,Z 488.456,A -85,B 0,C 180,E1 -7017.493,E2 -7017.493} C_VEL
LIN {X 0,Y 481.945,Z 488.454,A -85,B 0,C 180,E1 -7020,E2 -7020} C_VEL
LIN {X 0,Y 481.931,Z 488.456,A -85,B 0,C 180,E1 -7022.508,E2 -7022.508} C_VEL
LIN {X 0,Y 481.795,Z 488.471,A -85,B 0,C 180,E1 -7025.861,E2 -7025.861} C_VEL
LIN {X 0,Y 481.766,Z 488.476,A -85,B 0,C 180,E1 -7028.389,E2 -7028.389} C_VEL
LIN {X 0,Y 481.756,Z 488.476,A -85,B 0,C 180,E1 -7031.785,E2 -7031.785} C_VEL
LIN {X 0,Y 481.748,Z 488.478,A -85,B 0,C 180,E1 -7035.224,E2 -7035.224} C_VEL
LIN {X 0,Y 481.714,Z 488.487,A -85,B 0,C 180,E1 -7038.722,E2 -7038.722} C_VEL
LIN {X 0,Y 481.714,Z 488.549,A -85,B 0,C 180,E1 -7039.912,E2 -7039.912} C_VEL
LIN {X 0,Y 483.942,Z 496.44,A -85,B 0,C 180,E1 -7040.398,E2 -7040.398} C_VEL
LIN {X 0,Y 483.743,Z 507.25,A -85,B 0,C 180,E1 -7041.075,E2 -7041.075} C_VEL
LIN {X 0,Y 483.377,Z 517.94,A -85,B 0,C 180,E1 -7041.913,E2 -7041.913} C_VEL
LIN {X 0,Y 482.975,Z 528.049,A -85,B 0,C 180,E1 -7042.908,E2 -7042.908} C_VEL
LIN {X 0,Y 482.538,Z 537.559,A -85,B 0,C 180,E1 -7044.068,E2 -7044.068} C_VEL
LIN {X 0,Y 482.173,Z 545.963,A -85,B 0,C 180,E1 -7045.351,E2 -7045.351} C_VEL
LIN {X 0,Y 481.915,Z 552.684,A -85,B 0,C 180,E1 -7046.644,E2 -7046.644} C_VEL
LIN {X 0,Y 481.662,Z 557.65,A -85,B 0,C 180,E1 -7047.835,E2 -7047.835} C_VEL
LIN {X 0,Y 481.486,Z 562.275,A -85,B 0,C 180,E1 -7049.274,E2 -7049.274} C_VEL
LIN {X 0,Y 481.356,Z 565.602,A -85,B 0,C 180,E1 -7050.732,E2 -7050.732} C_VEL
LIN {X 0,Y 481.238,Z 567.571,A -85,B 0,C 180,E1 -7052.109,E2 -7052.109} C_VEL
LIN {X 0,Y 481.199,Z 568.493,A -85,B 0,C 180,E1 -7053.711,E2 -7053.711} C_VEL
LIN {X 0,Y 481.189,Z 568.149,A -85,B 0,C 180,E1 -7055.124,E2 -7055.124} C_VEL
LIN {X 0,Y 481.253,Z 566.343,A -85,B 0,C 180,E1 -7056.781,E2 -7056.781} C_VEL
LIN {X 0,Y 481.368,Z 563.049,A -85,B 0,C 180,E1 -7058.38,E2 -7058.38} C_VEL
LIN {X 0,Y 481.492,Z 559.496,A -85,B 0,C 180,E1 -7059.597,E2 -7059.597} C_VEL
LIN {X 0,Y 481.7,Z 553.962,A -85,B 0,C 180,E1 -7061.038,E2 -7061.038} C_VEL
LIN {X 0,Y 481.979,Z 547.154,A -85,B 0,C 180,E1 -7062.408,E2 -7062.408} C_VEL
LIN {X 0,Y 482.267,Z 540.302,A -85,B 0,C 180,E1 -7063.517,E2 -7063.517} C_VEL
LIN {X 0,Y 482.69,Z 530.575,A -85,B 0,C 180,E1 -7064.791,E2 -7064.791} C_VEL
LIN {X 0,Y 483.106,Z 520.572,A -85,B 0,C 180,E1 -7065.841,E2 -7065.841} C_VEL
LIN {X 0,Y 483.473,Z 510.082,A -85,B 0,C 180,E1 -7066.725,E2 -7066.725} C_VEL
LIN {X 0,Y 483.858,Z 498.279,A -85,B 0,C 180,E1 -7067.514,E2 -7067.514} C_VEL
LIN {X 0,Y 483.765,Z 496.075,A -85,B 0,C 180,E1 -7067.645,E2 -7067.645} C_VEL
LIN {X 0,Y 481.677,Z 488.488,A -85,B 0,C 180,E1 -7068.116,E2 -7068.116} C_VEL
LIN {X 0,Y 481.672,Z 488.489,A -85,B 0,C 180,E1 -7071.141,E2 -7071.141} C_VEL
LIN {X 0,Y 481.665,Z 488.486,A -85,B 0,C 180,E1 -7074.796,E2 -7074.796} C_VEL
LIN {X 0,Y 481.677,Z 488.487,A -85,B 0,C 180,E1 -7077.326,E2 -7077.326} C_VEL
LIN {X 0,Y 481.683,Z 488.484,A -85,B 0,C 180,E1 -7080.259,E2 -7080.259} C_VEL
LIN {X 0,Y 481.695,Z 488.483,A -85,B 0,C 180,E1 -7081.352,E2 -7081.352} C_VEL
LIN {X 0,Y 481.009,Z 488.568,A -85,B 0,C 180,E1 -7082.05,E2 -7082.05} C_VEL
LIN {X 0,Y 478.153,Z 488.927,A -85,B 0,C 180,E1 -7083.183,E2 -7083.183} C_VEL
LIN {X 0,Y 475.749,Z 489.225,A -85,B 0,C 180,E1 -7084.097,E2 -7084.097} C_VEL
LIN {X 0,Y 474.716,Z 489.354,A -85,B 0,C 180,E1 -7084.802,E2 -7084.802} C_VEL
LIN {X 0,Y 474.63,Z 489.362,A -85,B 0,C 180,E1 -7085.041,E2 -7085.041} C_VEL
LIN {X 0,Y 474.606,Z 489.369,A -85,B 0,C 180,E1 -7087.355,E2 -7087.355} C_VEL
LIN {X 0,Y 474.659,Z 489.361,A -85,B 0,C 180,E1 -7090.09,E2 -7090.09} C_VEL
LIN {X 0,Y 474.641,Z 489.361,A -85,B 0,C 180,E1 -7092.774,E2 -7092.774} C_VEL
LIN {X 0,Y 474.65,Z 489.361,A -85,B 0,C 180,E1 -7095.421,E2 -7095.421} C_VEL
LIN {X 0,Y 474.711,Z 489.354,A -85,B 0,C 180,E1 -7098.038,E2 -7098.038} C_VEL
LIN {X 0,Y 474.715,Z 489.353,A -85,B 0,C 180,E1 -7101.486,E2 -7101.486} C_VEL
LIN {X 0,Y 474.748,Z 489.348,A -85,B 0,C 180,E1 -7104.904,E2 -7104.904} C_VEL
LIN {X 0,Y 474.899,Z 489.33,A -85,B 0,C 180,E1 -7107.455,E2 -7107.455} C_VEL
LIN {X 0,Y 474.913,Z 489.328,A -85,B 0,C 180,E1 -7110,E2 -7110} C_VEL
LIN {X 0,Y 474.892,Z 489.33,A -85,B 0,C 180,E1 -7112.545,E2 -7112.545} C_VEL
LIN {X 0,Y 474.754,Z 489.348,A -85,B 0,C 180,E1 -7115.948,E2 -7115.948} C_VEL
LIN {X 0,Y 474.718,Z 489.352,A -85,B 0,C 180,E1 -7118.514,E2 -7118.514} C_VEL
LIN {X 0,Y 474.71,Z 489.354,A -85,B 0,C 180,E1 -7121.962,E2 -7121.962} C_VEL
LIN {X 0,Y 474.705,Z 489.354,A -85,B 0,C 180,E1 -7125.455,E2 -7125.455} C_VEL
LIN {X 0,Y 474.667,Z 489.36,A -85,B 0,C 180,E1 -7129.01,E2 -7129.01} C_VEL
LIN {X 0,Y 474.593,Z 489.368,A -85,B 0,C 180,E1 -7131.729,E2 -7131.729} C_VEL
LIN {X 0,Y 474.634,Z 489.362,A -85,B 0,C 180,E1 -7134.494,E2 -7134.494} C_VEL
LIN {X 0,Y 474.641,Z 489.362,A -85,B 0,C 180,E1 -7137.324,E2 -7137.324} C_VEL
LIN {X 0,Y 474.606,Z 489.366,A -85,B 0,C 180,E1 -7140.23,E2 -7140.23} C_VEL
LIN {X 0,Y 474.629,Z 489.364,A -85,B 0,C 180,E1 -7143.221,E2 -7143.221} C_VEL
LIN {X 0,Y 474.588,Z 489.368,A -85,B 0,C 180,E1 -7146.324,E2 -7146.324} C_VEL
LIN {X 0,Y 474.626,Z 489.364,A -85,B 0,C 180,E1 -7149.548,E2 -7149.548} C_VEL
LIN {X 0,Y 474.592,Z 489.368,A -85,B 0,C 180,E1 -7152.232,E2 -7152.232} C_VEL
LIN {X 0,Y 474.62,Z 489.365,A -85,B 0,C 180,E1 -7155.298,E2 -7155.298} C_VEL
LIN {X 0,Y 474.618,Z 489.364,A -85,B 0,C 180,E1 -7158.214,E2 -7158.214} C_VEL
LIN {X 0,Y 474.613,Z 489.365,A -85,B 0,C 180,E1 -7161.542,E2 -7161.542} C_VEL
LIN {X 0,Y 474.625,Z 489.364,A -85,B 0,C 180,E1 -7164.725,E2 -7164.725} C_VEL
LIN {X 0,Y 474.639,Z 489.363,A -85,B 0,C 180,E1 -7167.788,E2 -7167.788} C_VEL
LIN {X 0,Y 474.628,Z 489.365,A -85,B 0,C 180,E1 -7170.884,E2 -7170.884} C_VEL
LIN {X 0,Y 474.631,Z 489.363,A -85,B 0,C 180,E1 -7173.626,E2 -7173.626} C_VEL
LIN {X 0,Y 474.637,Z 489.362,A -85,B 0,C 180,E1 -7176.642,E2 -7176.642} C_VEL
LIN {X 0,Y 474.656,Z 489.361,A -85,B 0,C 180,E1 -7180.089,E2 -7180.089} C_VEL
LIN {X 0,Y 474.639,Z 489.363,A -85,B 0,C 180,E1 -7182.774,E2 -7182.774} C_VEL
LIN {X 0,Y 474.648,Z 489.361,A -85,B 0,C 180,E1 -7185.421,E2 -7185.421} C_VEL
LIN {X 0,Y 474.708,Z 489.354,A -85,B 0,C 180,E1 -7188.037,E2 -7188.037} C_VEL
LIN {X 0,Y 474.712,Z 489.353,A -85,B 0,C 180,E1 -7191.486,E2 -7191.486} C_VEL
LIN {X 0,Y 474.749,Z 489.35,A -85,B 0,C 180,E1 -7194.904,E2 -7194.904} C_VEL
LIN {X 0,Y 474.889,Z 489.331,A -85,B 0,C 180,E1 -7197.455,E2 -7197.455} C_VEL
LIN {X 0,Y 474.913,Z 489.328,A -85,B 0,C 180,E1 -7200,E2 -7200} C_VEL
LIN {X 0,Y 474.885,Z 489.333,A -85,B 0,C 180,E1 -7202.544,E2 -7202.544} C_VEL
LIN {X 0,Y 474.753,Z 489.348,A -85,B 0,C 180,E1 -7205.948,E2 -7205.948} C_VEL
LIN {X 0,Y 474.728,Z 489.352,A -85,B 0,C 180,E1 -7208.513,E2 -7208.513} C_VEL
LIN {X 0,Y 474.742,Z 489.35,A -85,B 0,C 180,E1 -7211.961,E2 -7211.961} C_VEL
LIN {X 0,Y 474.682,Z 489.357,A -85,B 0,C 180,E1 -7215.767,E2 -7215.767} C_VEL
LIN {X 0,Y 474.665,Z 489.362,A -85,B 0,C 180,E1 -7219.01,E2 -7219.01} C_VEL
LIN {X 0,Y 474.59,Z 489.369,A -85,B 0,C 180,E1 -7221.729,E2 -7221.729} C_VEL
LIN {X 0,Y 474.638,Z 489.362,A -85,B 0,C 180,E1 -7224.494,E2 -7224.494} C_VEL
LIN {X 0,Y 474.638,Z 489.362,A -85,B 0,C 180,E1 -7227.324,E2 -7227.324} C_VEL
LIN {X 0,Y 474.604,Z 489.366,A -85,B 0,C 180,E1 -7230.23,E2 -7230.23} C_VEL
LIN {X 0,Y 474.626,Z 489.363,A -85,B 0,C 180,E1 -7233.221,E2 -7233.221} C_VEL
LIN {X 0,Y 474.59,Z 489.368,A -85,B 0,C 180,E1 -7236.323,E2 -7236.323} C_VEL
LIN {X 0,Y 474.617,Z 489.366,A -85,B 0,C 180,E1 -7239.646,E2 -7239.646} C_VEL
LIN {X 0,Y 474.616,Z 489.368,A -85,B 0,C 180,E1 -7242.934,E2 -7242.934} C_VEL
LIN {X 0,Y 474.604,Z 489.365,A -85,B 0,C 180,E1 -7245.894,E2 -7245.894} C_VEL
LIN {X 0,Y 474.628,Z 489.361,A -85,B 0,C 180,E1 -7249.192,E2 -7249.192} C_VEL
LIN {X 0,Y 474.623,Z 489.368,A -85,B 0,C 180,E1 -7249.343,E2 -7249.343} C_VEL
LIN {X 0,Y 476.999,Z 501.307,A -85,B 0,C 180,E1 -7252.714,E2 -7252.714} C_VEL
LIN {X 0,Y 477.444,Z 505.868,A -85,B 0,C 180,E1 -7253.928,E2 -7253.928} C_VEL
LIN {X 0,Y 476.794,Z 517.969,A -85,B 0,C 180,E1 -7256.949,E2 -7256.949} C_VEL
LIN {X 0,Y 476.324,Z 530.076,A -85,B 0,C 180,E1 -7259.89,E2 -7259.89} C_VEL
LIN {X 0,Y 475.716,Z 545.229,A -85,B 0,C 180,E1 -7263.455,E2 -7263.455} C_VEL
LIN {X 0,Y 475.299,Z 558.32,A -85,B 0,C 180,E1 -7266.47,E2 -7266.47} C_VEL
LIN {X 0,Y 474.883,Z 573.453,A -85,B 0,C 180,E1 -7269.874,E2 -7269.874} C_VEL
LIN {X 0,Y 474.553,Z 588.586,A -85,B 0,C 180,E1 -7273.215,E2 -7273.215} C_VEL
LIN {X 0,Y 474.401,Z 595.704,A -85,B 0,C 180,E1 -7274.782,E2 -7274.782} C_VEL
LIN {X 0,Y 475.981,Z 611.776,A -85,B 0,C 180,E1 -7275.244,E2 -7275.244} C_VEL
LIN {X 0,Y 476.688,Z 619.287,A -85,B 0,C 180,E1 -7275.539,E2 -7275.539} C_VEL
LIN {X 0,Y 476.248,Z 631.748,A -85,B 0,C 180,E1 -7276.125,E2 -7276.125} C_VEL
LIN {X 0,Y 475.762,Z 643.8,A -85,B 0,C 180,E1 -7276.872,E2 -7276.872} C_VEL
LIN {X 0,Y 475.39,Z 654.243,A -85,B 0,C 180,E1 -7277.695,E2 -7277.695} C_VEL
LIN {X 0,Y 474.972,Z 664.517,A -85,B 0,C 180,E1 -7278.694,E2 -7278.694} C_VEL
LIN {X 0,Y 474.551,Z 673.536,A -85,B 0,C 180,E1 -7279.763,E2 -7279.763} C_VEL
LIN {X 0,Y 474.284,Z 682.38,A -85,B 0,C 180,E1 -7281.049,E2 -7281.049} C_VEL
LIN {X 0,Y 474.102,Z 689.452,A -85,B 0,C 180,E1 -7282.333,E2 -7282.333} C_VEL
LIN {X 0,Y 474.022,Z 695.371,A -85,B 0,C 180,E1 -7283.678,E2 -7283.678} C_VEL
LIN {X 0,Y 473.965,Z 699.581,A -85,B 0,C 180,E1 -7284.896,E2 -7284.896} C_VEL
LIN {X 0,Y 473.964,Z 701.932,A -85,B 0,C 180,E1 -7285.748,E2 -7285.748} C_VEL
LIN {X 0,Y 473.968,Z 703.841,A -85,B 0,C 180,E1 -7286.6,E2 -7286.6} C_VEL
LIN {X 0,Y 473.948,Z 705.27,A -85,B 0,C 180,E1 -7287.45,E2 -7287.45} C_VEL
LIN {X 0,Y 473.927,Z 706.279,A -85,B 0,C 180,E1 -7288.301,E2 -7288.301} C_VEL
LIN {X 0,Y 473.99,Z 707.093,A -85,B 0,C 180,E1 -7290,E2 -7290} C_VEL
LIN {X 0,Y 473.939,Z 706.19,A -85,B 0,C 180,E1 -7291.7,E2 -7291.7} C_VEL
LIN {X 0,Y 473.966,Z 705.132,A -85,B 0,C 180,E1 -7292.55,E2 -7292.55} C_VEL
LIN {X 0,Y 473.985,Z 703.656,A -85,B 0,C 180,E1 -7293.4,E2 -7293.4} C_VEL
LIN {X 0,Y 473.98,Z 700.568,A -85,B 0,C 180,E1 -7294.678,E2 -7294.678} C_VEL
LIN {X 0,Y 474.052,Z 696.41,A -85,B 0,C 180,E1 -7295.957,E2 -7295.957} C_VEL
LIN {X 0,Y 474.114,Z 690.022,A -85,B 0,C 180,E1 -7297.453,E2 -7297.453} C_VEL
LIN {X 0,Y 474.296,Z 683.07,A -85,B 0,C 180,E1 -7298.736,E2 -7298.736} C_VEL
LIN {X 0,Y 474.499,Z 674.46,A -85,B 0,C 180,E1 -7300.023,E2 -7300.023} C_VEL
LIN {X 0,Y 474.938,Z 664.663,A -85,B 0,C 180,E1 -7301.199,E2 -7301.199} C_VEL
LIN {X 0,Y 475.307,Z 655.375,A -85,B 0,C 180,E1 -7302.116,E2 -7302.116} C_VEL
LIN {X 0,Y 475.668,Z 644.151,A -85,B 0,C 180,E1 -7303.022,E2 -7303.022} C_VEL
LIN {X 0,Y 476.132,Z 632.474,A -85,B 0,C 180,E1 -7303.77,E2 -7303.77} C_VEL
LIN {X 0,Y 476.616,Z 619.195,A -85,B 0,C 180,E1 -7304.409,E2 -7304.409} C_VEL
LIN {X 0,Y 476.088,Z 613.084,A -85,B 0,C 180,E1 -7304.657,E2 -7304.657} C_VEL
LIN {X 0,Y 475.162,Z 603.55,A -85,B 0,C 180,E1 -7304.974,E2 -7304.974} C_VEL
LIN {X 0,Y 474.392,Z 594.164,A -85,B 0,C 180,E1 -7305.219,E2 -7305.219} C_VEL
LIN {X 0,Y 474.643,Z 579.419,A -85,B 0,C 180,E1 -7308.367,E2 -7308.367} C_VEL
LIN {X 0,Y 474.907,Z 563.932,A -85,B 0,C 180,E1 -7311.714,E2 -7311.714} C_VEL
LIN {X 0,Y 475.263,Z 548.302,A -85,B 0,C 180,E1 -7315.16,E2 -7315.16} C_VEL
LIN {X 0,Y 475.542,Z 534.778,A -85,B 0,C 180,E1 -7318.225,E2 -7318.225} C_VEL
LIN {X 0,Y 476.002,Z 521.36,A -85,B 0,C 180,E1 -7321.363,E2 -7321.363} C_VEL
LIN {X 0,Y 476.468,Z 507.908,A -85,B 0,C 180,E1 -7324.657,E2 -7324.657} C_VEL
LIN {X 0,Y 476.776,Z 502.099,A -85,B 0,C 180,E1 -7326.131,E2 -7326.131} C_VEL
LIN {X 0,Y 476.146,Z 497.055,A -85,B 0,C 180,E1 -7327.507,E2 -7327.507} C_VEL
LIN {X 0,Y 474.66,Z 489.36,A -85,B 0,C 180,E1 -7329.746,E2 -7329.746} C_VEL
LIN {X 0,Y 474.618,Z 489.368,A -85,B 0,C 180,E1 -7332.934,E2 -7332.934} C_VEL
LIN {X 0,Y 474.612,Z 489.37,A -85,B 0,C 180,E1 -7335.895,E2 -7335.895} C_VEL
LIN {X 0,Y 474.631,Z 489.366,A -85,B 0,C 180,E1 -7339.041,E2 -7339.041} C_VEL
LIN {X 0,Y 474.611,Z 489.365,A -85,B 0,C 180,E1 -7341.705,E2 -7341.705} C_VEL
LIN {X 0,Y 474.623,Z 489.366,A -85,B 0,C 180,E1 -7344.726,E2 -7344.726} C_VEL
LIN {X 0,Y 474.638,Z 489.361,A -85,B 0,C 180,E1 -7347.788,E2 -7347.788} C_VEL
LIN {X 0,Y 474.627,Z 489.362,A -85,B 0,C 180,E1 -7350.885,E2 -7350.885} C_VEL
LIN {X 0,Y 474.657,Z 489.359,A -85,B 0,C 180,E1 -7353.628,E2 -7353.628} C_VEL
LIN {X 0,Y 474.638,Z 489.361,A -85,B 0,C 180,E1 -7356.642,E2 -7356.642} C_VEL
LIN {X 0,Y 474.658,Z 489.361,A -85,B 0,C 180,E1 -7360.09,E2 -7360.09} C_VEL
LIN {X 0,Y 474.642,Z 489.362,A -85,B 0,C 180,E1 -7362.774,E2 -7362.774} C_VEL
LIN {X 0,Y 474.651,Z 489.358,A -85,B 0,C 180,E1 -7365.421,E2 -7365.421} C_VEL
LIN {X 0,Y 474.709,Z 489.353,A -85,B 0,C 180,E1 -7368.038,E2 -7368.038} C_VEL
LIN {X 0,Y 474.731,Z 489.349,A -85,B 0,C 180,E1 -7371.487,E2 -7371.487} C_VEL
LIN {X 0,Y 474.783,Z 489.344,A -85,B 0,C 180,E1 -7374.053,E2 -7374.053} C_VEL
LIN {X 0,Y 474.888,Z 489.332,A -85,B 0,C 180,E1 -7377.456,E2 -7377.456} C_VEL
LIN {X 0,Y 474.916,Z 489.329,A -85,B 0,C 180,E1 -7380,E2 -7380} C_VEL
LIN {X 0,Y 474.897,Z 489.332,A -85,B 0,C 180,E1 -7382.545,E2 -7382.545} C_VEL
LIN {X 0,Y 474.756,Z 489.347,A -85,B 0,C 180,E1 -7385.948,E2 -7385.948} C_VEL
LIN {X 0,Y 474.731,Z 489.351,A -85,B 0,C 180,E1 -7388.514,E2 -7388.514} C_VEL
LIN {X 0,Y 474.709,Z 489.355,A -85,B 0,C 180,E1 -7391.963,E2 -7391.963} C_VEL
LIN {X 0,Y 474.705,Z 489.356,A -85,B 0,C 180,E1 -7395.456,E2 -7395.456} C_VEL
LIN {X 0,Y 474.674,Z 489.364,A -85,B 0,C 180,E1 -7399.01,E2 -7399.01} C_VEL
LIN {X 0,Y 474.683,Z 489.364,A -85,B 0,C 180,E1 -7399.684,E2 -7399.684} C_VEL
LIN {X 0,Y 477.18,Z 498.36,A -85,B 0,C 180,E1 -7400.25,E2 -7400.25} C_VEL
LIN {X 0,Y 476.889,Z 509.085,A -85,B 0,C 180,E1 -7400.94,E2 -7400.94} C_VEL
LIN {X 0,Y 476.471,Z 520.171,A -85,B 0,C 180,E1 -7401.844,E2 -7401.844} C_VEL
LIN {X 0,Y 476.026,Z 530.642,A -85,B 0,C 180,E1 -7402.917,E2 -7402.917} C_VEL
LIN {X 0,Y 475.623,Z 539.163,A -85,B 0,C 180,E1 -7403.995,E2 -7403.995} C_VEL
LIN {X 0,Y 475.269,Z 546.668,A -85,B 0,C 180,E1 -7405.16,E2 -7405.16} C_VEL
LIN {X 0,Y 474.949,Z 554.002,A -85,B 0,C 180,E1 -7406.592,E2 -7406.592} C_VEL
LIN {X 0,Y 474.698,Z 558.906,A -85,B 0,C 180,E1 -7407.799,E2 -7407.799} C_VEL
LIN {X 0,Y 474.503,Z 563.483,A -85,B 0,C 180,E1 -7409.26,E2 -7409.26} C_VEL
LIN {X 0,Y 474.34,Z 566.772,A -85,B 0,C 180,E1 -7410.756,E2 -7410.756} C_VEL
LIN {X 0,Y 474.197,Z 568.843,A -85,B 0,C 180,E1 -7412.35,E2 -7412.35} C_VEL
LIN {X 0,Y 474.18,Z 569.545,A -85,B 0,C 180,E1 -7413.901,E2 -7413.901} C_VEL
LIN {X 0,Y 474.164,Z 569.011,A -85,B 0,C 180,E1 -7415.392,E2 -7415.392} C_VEL
LIN {X 0,Y 474.233,Z 567.309,A -85,B 0,C 180,E1 -7416.844,E2 -7416.844} C_VEL
LIN {X 0,Y 474.386,Z 563.95,A -85,B 0,C 180,E1 -7418.48,E2 -7418.48} C_VEL
LIN {X 0,Y 474.563,Z 559.021,A -85,B 0,C 180,E1 -7420.107,E2 -7420.107} C_VEL
LIN {X 0,Y 474.805,Z 553.103,A -85,B 0,C 180,E1 -7421.541,E2 -7421.541} C_VEL
LIN {X 0,Y 475.105,Z 546.096,A -85,B 0,C 180,E1 -7422.88,E2 -7422.88} C_VEL
LIN {X 0,Y 475.531,Z 537.786,A -85,B 0,C 180,E1 -7424.145,E2 -7424.145} C_VEL
LIN {X 0,Y 475.921,Z 528.463,A -85,B 0,C 180,E1 -7425.29,E2 -7425.29} C_VEL
LIN {X 0,Y 476.332,Z 518.318,A -85,B 0,C 180,E1 -7426.301,E2 -7426.301} C_VEL
LIN {X 0,Y 476.732,Z 507.356,A -85,B 0,C 180,E1 -7427.174,E2 -7427.174} C_VEL
LIN {X 0,Y 477.046,Z 498.108,A -85,B 0,C 180,E1 -7427.769,E2 -7427.769} C_VEL
LIN {X 0,Y 474.634,Z 489.364,A -85,B 0,C 180,E1 -7428.329,E2 -7428.329} C_VEL
LIN {X 0,Y 474.612,Z 489.366,A -85,B 0,C 180,E1 -7431.705,E2 -7431.705} C_VEL
LIN {X 0,Y 474.627,Z 489.362,A -85,B 0,C 180,E1 -7434.726,E2 -7434.726} C_VEL
LIN {X 0,Y 474.641,Z 489.362,A -85,B 0,C 180,E1 -7437.788,E2 -7437.788} C_VEL
LIN {X 0,Y 474.627,Z 489.363,A -85,B 0,C 180,E1 -7440.885,E2 -7440.885} C_VEL
LIN {X 0,Y 474.634,Z 489.363,A -85,B 0,C 180,E1 -7443.627,E2 -7443.627} C_VEL
LIN {X 0,Y 474.63,Z 489.362,A -85,B 0,C 180,E1 -7445.041,E2 -7445.041} C_VEL
LIN {X 0,Y 473.954,Z 489.45,A -85,B 0,C 180,E1 -7445.749,E2 -7445.749} C_VEL
LIN {X 0,Y 471.085,Z 489.804,A -85,B 0,C 180,E1 -7446.898,E2 -7446.898} C_VEL
LIN {X 0,Y 468.675,Z 490.104,A -85,B 0,C 180,E1 -7447.825,E2 -7447.825} C_VEL
LIN {X 0,Y 467.661,Z 490.231,A -85,B 0,C 180,E1 -7448.541,E2 -7448.541} C_VEL
LIN {X 0,Y 467.588,Z 490.241,A -85,B 0,C 180,E1 -7448.783,E2 -7448.783} C_VEL
LIN {X 0,Y 467.629,Z 490.237,A -85,B 0,C 180,E1 -7451.602,E2 -7451.602} C_VEL
LIN {X 0,Y 467.644,Z 490.232,A -85,B 0,C 180,E1 -7454.305,E2 -7454.305} C_VEL
LIN {X 0,Y 467.662,Z 490.233,A -85,B 0,C 180,E1 -7457.855,E2 -7457.855} C_VEL
LIN {X 0,Y 467.674,Z 490.23,A -85,B 0,C 180,E1 -7461.357,E2 -7461.357} C_VEL
LIN {X 0,Y 467.718,Z 490.225,A -85,B 0,C 180,E1 -7463.962,E2 -7463.962} C_VEL
LIN {X 0,Y 467.865,Z 490.206,A -85,B 0,C 180,E1 -7467.417,E2 -7467.417} C_VEL
LIN {X 0,Y 467.882,Z 490.204,A -85,B 0,C 180,E1 -7470,E2 -7470} C_VEL
LIN {X 0,Y 467.857,Z 490.207,A -85,B 0,C 180,E1 -7472.583,E2 -7472.583} C_VEL
LIN {X 0,Y 467.717,Z 490.224,A -85,B 0,C 180,E1 -7476.038,E2 -7476.038} C_VEL
LIN {X 0,Y 467.676,Z 490.23,A -85,B 0,C 180,E1 -7478.643,E2 -7478.643} C_VEL
LIN {X 0,Y 467.662,Z 490.231,A -85,B 0,C 180,E1 -7482.145,E2 -7482.145} C_VEL
LIN {X 0,Y 467.644,Z 490.234,A -85,B 0,C 180,E1 -7485.695,E2 -7485.695} C_VEL
LIN {X 0,Y 467.626,Z 490.239,A -85,B 0,C 180,E1 -7489.308,E2 -7489.308} C_VEL
LIN {X 0,Y 467.539,Z 490.247,A -85,B 0,C 180,E1 -7492.074,E2 -7492.074} C_VEL
LIN {X 0,Y 467.574,Z 490.242,A -85,B 0,C 180,E1 -7494.889,E2 -7494.889} C_VEL
LIN {X 0,Y 467.584,Z 490.241,A -85,B 0,C 180,E1 -7497.771,E2 -7497.771} C_VEL
LIN {X 0,Y 467.572,Z 490.244,A -85,B 0,C 180,E1 -7501.044,E2 -7501.044} C_VEL
LIN {X 0,Y 467.581,Z 490.242,A -85,B 0,C 180,E1 -7504.24,E2 -7504.24} C_VEL
LIN {X 0,Y 467.547,Z 490.249,A -85,B 0,C 180,E1 -7507.185,E2 -7507.185} C_VEL
LIN {X 0,Y 467.562,Z 490.244,A -85,B 0,C 180,E1 -7510.266,E2 -7510.266} C_VEL
LIN {X 0,Y 467.55,Z 490.244,A -85,B 0,C 180,E1 -7513.745,E2 -7513.745} C_VEL
LIN {X 0,Y 467.552,Z 490.246,A -85,B 0,C 180,E1 -7516.254,E2 -7516.254} C_VEL
LIN {X 0,Y 467.574,Z 490.241,A -85,B 0,C 180,E1 -7519.734,E2 -7519.734} C_VEL
LIN {X 0,Y 467.545,Z 490.246,A -85,B 0,C 180,E1 -7522.815,E2 -7522.815} C_VEL
LIN {X 0,Y 467.589,Z 490.239,A -85,B 0,C 180,E1 -7526.212,E2 -7526.212} C_VEL
LIN {X 0,Y 467.573,Z 490.244,A -85,B 0,C 180,E1 -7529.266,E2 -7529.266} C_VEL
LIN {X 0,Y 467.632,Z 490.235,A -85,B 0,C 180,E1 -7532.463,E2 -7532.463} C_VEL
LIN {X 0,Y 467.582,Z 490.242,A -85,B 0,C 180,E1 -7535.111,E2 -7535.111} C_VEL
LIN {X 0,Y 467.537,Z 490.245,A -85,B 0,C 180,E1 -7537.926,E2 -7537.926} C_VEL
LIN {X 0,Y 467.624,Z 490.237,A -85,B 0,C 180,E1 -7540.692,E2 -7540.692} C_VEL
LIN {X 0,Y 467.642,Z 490.233,A -85,B 0,C 180,E1 -7544.305,E2 -7544.305} C_VEL
LIN {X 0,Y 467.659,Z 490.232,A -85,B 0,C 180,E1 -7547.854,E2 -7547.854} C_VEL
LIN {X 0,Y 467.67,Z 490.23,A -85,B 0,C 180,E1 -7551.357,E2 -7551.357} C_VEL
LIN {X 0,Y 467.721,Z 490.224,A -85,B 0,C 180,E1 -7553.962,E2 -7553.962} C_VEL
LIN {X 0,Y 467.855,Z 490.207,A -85,B 0,C 180,E1 -7557.417,E2 -7557.417} C_VEL
LIN {X 0,Y 467.883,Z 490.204,A -85,B 0,C 180,E1 -7560,E2 -7560} C_VEL
LIN {X 0,Y 467.849,Z 490.21,A -85,B 0,C 180,E1 -7562.583,E2 -7562.583} C_VEL
LIN {X 0,Y 467.716,Z 490.225,A -85,B 0,C 180,E1 -7566.038,E2 -7566.038} C_VEL
LIN {X 0,Y 467.682,Z 490.232,A -85,B 0,C 180,E1 -7568.643,E2 -7568.643} C_VEL
LIN {X 0,Y 467.676,Z 490.229,A -85,B 0,C 180,E1 -7572.368,E2 -7572.368} C_VEL
LIN {X 0,Y 467.651,Z 490.233,A -85,B 0,C 180,E1 -7575.885,E2 -7575.885} C_VEL
LIN {X 0,Y 467.624,Z 490.236,A -85,B 0,C 180,E1 -7579.308,E2 -7579.308} C_VEL
LIN {X 0,Y 467.536,Z 490.248,A -85,B 0,C 180,E1 -7582.074,E2 -7582.074} C_VEL
LIN {X 0,Y 467.585,Z 490.244,A -85,B 0,C 180,E1 -7584.888,E2 -7584.888} C_VEL
LIN {X 0,Y 467.581,Z 490.242,A -85,B 0,C 180,E1 -7587.771,E2 -7587.771} C_VEL
LIN {X 0,Y 467.57,Z 490.245,A -85,B 0,C 180,E1 -7591.045,E2 -7591.045} C_VEL
LIN {X 0,Y 467.578,Z 490.244,A -85,B 0,C 180,E1 -7594.24,E2 -7594.24} C_VEL
LIN {X 0,Y 467.549,Z 490.246,A -85,B 0,C 180,E1 -7597.186,E2 -7597.186} C_VEL
LIN {X 0,Y 467.575,Z 490.244,A -85,B 0,C 180,E1 -7600.265,E2 -7600.265} C_VEL
LIN {X 0,Y 467.588,Z 490.241,A -85,B 0,C 180,E1 -7602.567,E2 -7602.567} C_VEL
LIN {X 0,Y 467.567,Z 490.24,A -85,B 0,C 180,E1 -7605.052,E2 -7605.052} C_VEL
LIN {X 0,Y 467.577,Z 490.239,A -85,B 0,C 180,E1 -7608.597,E2 -7608.597} C_VEL
LIN {X 0,Y 467.614,Z 490.436,A -85,B 0,C 180,E1 -7609.101,E2 -7609.101} C_VEL
LIN {X 0,Y 469.945,Z 501.99,A -85,B 0,C 180,E1 -7612.43,E2 -7612.43} C_VEL
LIN {X 0,Y 470.508,Z 506.894,A -85,B 0,C 180,E1 -7613.765,E2 -7613.765} C_VEL
LIN {X 0,Y 469.948,Z 517.258,A -85,B 0,C 180,E1 -7616.404,E2 -7616.404} C_VEL
LIN {X 0,Y 469.324,Z 531.356,A -85,B 0,C 180,E1 -7619.891,E2 -7619.891} C_VEL
LIN {X 0,Y 468.67,Z 546.47,A -85,B 0,C 180,E1 -7623.505,E2 -7623.505} C_VEL
LIN {X 0,Y 468.205,Z 559.973,A -85,B 0,C 180,E1 -7626.655,E2 -7626.655} C_VEL
LIN {X 0,Y 467.804,Z 573.603,A -85,B 0,C 180,E1 -7629.785,E2 -7629.785} C_VEL
LIN {X 0,Y 467.495,Z 587.653,A -85,B 0,C 180,E1 -7632.953,E2 -7632.953} C_VEL
LIN {X 0,Y 467.337,Z 594.938,A -85,B 0,C 180,E1 -7634.574,E2 -7634.574} C_VEL
LIN {X 0,Y 468.679,Z 609.283,A -85,B 0,C 180,E1 -7634.967,E2 -7634.967} C_VEL
LIN {X 0,Y 469.741,Z 619.535,A -85,B 0,C 180,E1 -7635.376,E2 -7635.376} C_VEL
LIN {X 0,Y 469.237,Z 632.69,A -85,B 0,C 180,E1 -7636.024,E2 -7636.024} C_VEL
LIN {X 0,Y 468.728,Z 644.235,A -85,B 0,C 180,E1 -7636.782,E2 -7636.782} C_VEL
LIN {X 0,Y 468.311,Z 655.535,A -85,B 0,C 180,E1 -7637.721,E2 -7637.721} C_VEL
LIN {X 0,Y 467.866,Z 665.474,A -85,B 0,C 180,E1 -7638.739,E2 -7638.739} C_VEL
LIN {X 0,Y 467.452,Z 674.159,A -85,B 0,C 180,E1 -7639.825,E2 -7639.825} C_VEL
LIN {X 0,Y 467.178,Z 682.632,A -85,B 0,C 180,E1 -7641.13,E2 -7641.13} C_VEL
LIN {X 0,Y 467.012,Z 689.474,A -85,B 0,C 180,E1 -7642.434,E2 -7642.434} C_VEL
LIN {X 0,Y 466.987,Z 695.765,A -85,B 0,C 180,E1 -7643.953,E2 -7643.953} C_VEL
LIN {X 0,Y 466.916,Z 699.833,A -85,B 0,C 180,E1 -7645.251,E2 -7645.251} C_VEL
LIN {X 0,Y 466.924,Z 702.836,A -85,B 0,C 180,E1 -7646.548,E2 -7646.548} C_VEL
LIN {X 0,Y 466.907,Z 704.265,A -85,B 0,C 180,E1 -7647.412,E2 -7647.412} C_VEL
LIN {X 0,Y 466.893,Z 705.269,A -85,B 0,C 180,E1 -7648.275,E2 -7648.275} C_VEL
LIN {X 0,Y 466.979,Z 706.08,A -85,B 0,C 180,E1 -7650,E2 -7650} C_VEL
LIN {X 0,Y 466.908,Z 705.16,A -85,B 0,C 180,E1 -7651.725,E2 -7651.725} C_VEL
LIN {X 0,Y 466.928,Z 704.095,A -85,B 0,C 180,E1 -7652.588,E2 -7652.588} C_VEL
LIN {X 0,Y 466.941,Z 702.612,A -85,B 0,C 180,E1 -7653.452,E2 -7653.452} C_VEL
LIN {X 0,Y 466.94,Z 699.51,A -85,B 0,C 180,E1 -7654.749,E2 -7654.749} C_VEL
LIN {X 0,Y 466.997,Z 695.334,A -85,B 0,C 180,E1 -7656.047,E2 -7656.047} C_VEL
LIN {X 0,Y 467.082,Z 688.924,A -85,B 0,C 180,E1 -7657.566,E2 -7657.566} C_VEL
LIN {X 0,Y 467.201,Z 681.942,A -85,B 0,C 180,E1 -7658.87,E2 -7658.87} C_VEL
LIN {X 0,Y 467.454,Z 673.319,A -85,B 0,C 180,E1 -7660.175,E2 -7660.175} C_VEL
LIN {X 0,Y 467.867,Z 663.498,A -85,B 0,C 180,E1 -7661.371,E2 -7661.371} C_VEL
LIN {X 0,Y 468.314,Z 652.911,A -85,B 0,C 180,E1 -7662.418,E2 -7662.418} C_VEL
LIN {X 0,Y 468.785,Z 641.513,A -85,B 0,C 180,E1 -7663.327,E2 -7663.327} C_VEL
LIN {X 0,Y 469.302,Z 629.32,A -85,B 0,C 180,E1 -7664.085,E2 -7664.085} C_VEL
LIN {X 0,Y 469.666,Z 618.028,A -85,B 0,C 180,E1 -7664.627,E2 -7664.627} C_VEL
LIN {X 0,Y 468.447,Z 607.255,A -85,B 0,C 180,E1 -7665.055,E2 -7665.055} C_VEL
LIN {X 0,Y 467.306,Z 593.014,A -85,B 0,C 180,E1 -7665.455,E2 -7665.455} C_VEL
LIN {X 0,Y 467.562,Z 579.473,A -85,B 0,C 180,E1 -7668.401,E2 -7668.401} C_VEL
LIN {X 0,Y 467.805,Z 564.726,A -85,B 0,C 180,E1 -7671.646,E2 -7671.646} C_VEL
LIN {X 0,Y 468.149,Z 550.417,A -85,B 0,C 180,E1 -7674.857,E2 -7674.857} C_VEL
LIN {X 0,Y 468.489,Z 537.873,A -85,B 0,C 180,E1 -7677.738,E2 -7677.738} C_VEL
LIN {X 0,Y 468.919,Z 524.194,A -85,B 0,C 180,E1 -7680.984,E2 -7680.984} C_VEL
LIN {X 0,Y 469.375,Z 511.558,A -85,B 0,C 180,E1 -7684.113,E2 -7684.113} C_VEL
LIN {X 0,Y 469.792,Z 502.756,A -85,B 0,C 180,E1 -7686.387,E2 -7686.387} C_VEL
LIN {X 0,Y 468.722,Z 495.946,A -85,B 0,C 180,E1 -7688.317,E2 -7688.317} C_VEL
LIN {X 0,Y 467.611,Z 490.239,A -85,B 0,C 180,E1 -7690.075,E2 -7690.075} C_VEL
LIN {X 0,Y 467.589,Z 490.245,A -85,B 0,C 180,E1 -7692.567,E2 -7692.567} C_VEL
LIN {X 0,Y 467.573,Z 490.248,A -85,B 0,C 180,E1 -7695.053,E2 -7695.053} C_VEL
LIN {X 0,Y 467.592,Z 490.246,A -85,B 0,C 180,E1 -7697.44,E2 -7697.44} C_VEL
LIN {X 0,Y 467.585,Z 490.243,A -85,B 0,C 180,E1 -7700.855,E2 -7700.855} C_VEL
LIN {X 0,Y 467.56,Z 490.244,A -85,B 0,C 180,E1 -7704.262,E2 -7704.262} C_VEL
LIN {X 0,Y 467.582,Z 490.244,A -85,B 0,C 180,E1 -7707.322,E2 -7707.322} C_VEL
LIN {X 0,Y 467.573,Z 490.24,A -85,B 0,C 180,E1 -7710.668,E2 -7710.668} C_VEL
LIN {X 0,Y 467.616,Z 490.235,A -85,B 0,C 180,E1 -7713.2,E2 -7713.2} C_VEL
LIN {X 0,Y 467.594,Z 490.239,A -85,B 0,C 180,E1 -7716.469,E2 -7716.469} C_VEL
LIN {X 0,Y 467.626,Z 490.236,A -85,B 0,C 180,E1 -7719.777,E2 -7719.777} C_VEL
LIN {X 0,Y 467.602,Z 490.239,A -85,B 0,C 180,E1 -7722.507,E2 -7722.507} C_VEL
LIN {X 0,Y 467.609,Z 490.235,A -85,B 0,C 180,E1 -7725.197,E2 -7725.197} C_VEL
LIN {X 0,Y 467.66,Z 490.231,A -85,B 0,C 180,E1 -7727.855,E2 -7727.855} C_VEL
LIN {X 0,Y 467.684,Z 490.227,A -85,B 0,C 180,E1 -7731.357,E2 -7731.357} C_VEL
LIN {X 0,Y 467.748,Z 490.221,A -85,B 0,C 180,E1 -7733.963,E2 -7733.963} C_VEL
LIN {X 0,Y 467.852,Z 490.209,A -85,B 0,C 180,E1 -7737.417,E2 -7737.417} C_VEL
LIN {X 0,Y 467.886,Z 490.205,A -85,B 0,C 180,E1 -7740,E2 -7740} C_VEL
LIN {X 0,Y 467.863,Z 490.208,A -85,B 0,C 180,E1 -7742.583,E2 -7742.583} C_VEL
LIN {X 0,Y 467.719,Z 490.223,A -85,B 0,C 180,E1 -7746.038,E2 -7746.038} C_VEL
LIN {X 0,Y 467.685,Z 490.228,A -85,B 0,C 180,E1 -7748.643,E2 -7748.643} C_VEL
LIN {X 0,Y 467.661,Z 490.235,A -85,B 0,C 180,E1 -7752.146,E2 -7752.146} C_VEL
LIN {X 0,Y 467.644,Z 490.237,A -85,B 0,C 180,E1 -7755.695,E2 -7755.695} C_VEL
LIN {X 0,Y 467.658,Z 490.238,A -85,B 0,C 180,E1 -7759.421,E2 -7759.421} C_VEL
LIN {X 0,Y 470.371,Z 500.404,A -85,B 0,C 180,E1 -7760.1,E2 -7760.1} C_VEL
LIN {X 0,Y 470.058,Z 510.906,A -85,B 0,C 180,E1 -7760.8,E2 -7760.8} C_VEL
LIN {X 0,Y 469.581,Z 522.067,A -85,B 0,C 180,E1 -7761.742,E2 -7761.742} C_VEL
LIN {X 0,Y 469.112,Z 532.202,A -85,B 0,C 180,E1 -7762.809,E2 -7762.809} C_VEL
LIN {X 0,Y 468.702,Z 540.49,A -85,B 0,C 180,E1 -7763.882,E2 -7763.882} C_VEL
LIN {X 0,Y 468.322,Z 547.968,A -85,B 0,C 180,E1 -7765.07,E2 -7765.07} C_VEL
LIN {X 0,Y 467.984,Z 555.316,A -85,B 0,C 180,E1 -7766.537,E2 -7766.537} C_VEL
LIN {X 0,Y 467.716,Z 560.17,A -85,B 0,C 180,E1 -7767.763,E2 -7767.763} C_VEL
LIN {X 0,Y 467.504,Z 564.874,A -85,B 0,C 180,E1 -7769.317,E2 -7769.317} C_VEL
LIN {X 0,Y 467.3,Z 568.266,A -85,B 0,C 180,E1 -7770.989,E2 -7770.989} C_VEL
LIN {X 0,Y 467.17,Z 570.11,A -85,B 0,C 180,E1 -7772.599,E2 -7772.599} C_VEL
LIN {X 0,Y 467.157,Z 570.564,A -85,B 0,C 180,E1 -7774.164,E2 -7774.164} C_VEL
LIN {X 0,Y 467.159,Z 569.788,A -85,B 0,C 180,E1 -7775.67,E2 -7775.67} C_VEL
LIN {X 0,Y 467.241,Z 567.884,A -85,B 0,C 180,E1 -7777.136,E2 -7777.136} C_VEL
LIN {X 0,Y 467.376,Z 564.897,A -85,B 0,C 180,E1 -7778.562,E2 -7778.562} C_VEL
LIN {X 0,Y 467.54,Z 560.835,A -85,B 0,C 180,E1 -7779.948,E2 -7779.948} C_VEL
LIN {X 0,Y 467.773,Z 555.298,A -85,B 0,C 180,E1 -7781.382,E2 -7781.382} C_VEL
LIN {X 0,Y 468.11,Z 548.104,A -85,B 0,C 180,E1 -7782.82,E2 -7782.82} C_VEL
LIN {X 0,Y 468.528,Z 540.181,A -85,B 0,C 180,E1 -7784.085,E2 -7784.085} C_VEL
LIN {X 0,Y 468.952,Z 530.613,A -85,B 0,C 180,E1 -7785.315,E2 -7785.315} C_VEL
LIN {X 0,Y 469.421,Z 520.248,A -85,B 0,C 180,E1 -7786.382,E2 -7786.382} C_VEL
LIN {X 0,Y 469.828,Z 509.858,A -85,B 0,C 180,E1 -7787.246,E2 -7787.246} C_VEL
LIN {X 0,Y 470.135,Z 500.619,A -85,B 0,C 180,E1 -7787.868,E2 -7787.868} C_VEL
LIN {X 0,Y 469.541,Z 497.244,A -85,B 0,C 180,E1 -7788.091,E2 -7788.091} C_VEL
LIN {X 0,Y 467.591,Z 490.24,A -85,B 0,C 180,E1 -7788.562,E2 -7788.562} C_VEL
LIN {X 0,Y 467.567,Z 490.244,A -85,B 0,C 180,E1 -7791.955,E2 -7791.955} C_VEL
LIN {X 0,Y 467.568,Z 490.244,A -85,B 0,C 180,E1 -7795.167,E2 -7795.167} C_VEL
LIN {X 0,Y 467.588,Z 490.241,A -85,B 0,C 180,E1 -7798.26,E2 -7798.26} C_VEL
LIN {X 0,Y 467.579,Z 490.243,A -85,B 0,C 180,E1 -7801.25,E2 -7801.25} C_VEL
LIN {X 0,Y 467.594,Z 490.241,A -85,B 0,C 180,E1 -7804.159,E2 -7804.159} C_VEL
LIN {X 0,Y 467.582,Z 490.241,A -85,B 0,C 180,E1 -7806.996,E2 -7806.996} C_VEL
LIN {X 0,Y 467.588,Z 490.241,A -85,B 0,C 180,E1 -7808.783,E2 -7808.783} C_VEL
LIN {X 0,Y 466.947,Z 490.324,A -85,B 0,C 180,E1 -7809.503,E2 -7809.503} C_VEL
LIN {X 0,Y 464.094,Z 490.679,A -85,B 0,C 180,E1 -7810.672,E2 -7810.672} C_VEL
LIN {X 0,Y 461.666,Z 490.98,A -85,B 0,C 180,E1 -7811.614,E2 -7811.614} C_VEL
LIN {X 0,Y 460.625,Z 491.107,A -85,B 0,C 180,E1 -7812.342,E2 -7812.342} C_VEL
LIN {X 0,Y 460.543,Z 491.116,A -85,B 0,C 180,E1 -7812.589,E2 -7812.589} C_VEL
LIN {X 0,Y 460.569,Z 491.117,A -85,B 0,C 180,E1 -7814.965,E2 -7814.965} C_VEL
LIN {X 0,Y 460.616,Z 491.108,A -85,B 0,C 180,E1 -7818.559,E2 -7818.559} C_VEL
LIN {X 0,Y 460.624,Z 491.109,A -85,B 0,C 180,E1 -7821.224,E2 -7821.224} C_VEL
LIN {X 0,Y 460.683,Z 491.102,A -85,B 0,C 180,E1 -7823.87,E2 -7823.87} C_VEL
LIN {X 0,Y 460.806,Z 491.086,A -85,B 0,C 180,E1 -7827.377,E2 -7827.377} C_VEL
LIN {X 0,Y 460.852,Z 491.08,A -85,B 0,C 180,E1 -7830,E2 -7830} C_VEL
LIN {X 0,Y 460.797,Z 491.086,A -85,B 0,C 180,E1 -7832.622,E2 -7832.622} C_VEL
LIN {X 0,Y 460.682,Z 491.1,A -85,B 0,C 180,E1 -7836.13,E2 -7836.13} C_VEL
LIN {X 0,Y 460.626,Z 491.109,A -85,B 0,C 180,E1 -7838.776,E2 -7838.776} C_VEL
LIN {X 0,Y 460.619,Z 491.108,A -85,B 0,C 180,E1 -7842.445,E2 -7842.445} C_VEL
LIN {X 0,Y 460.606,Z 491.111,A -85,B 0,C 180,E1 -7845.997,E2 -7845.997} C_VEL
LIN {X 0,Y 460.573,Z 491.114,A -85,B 0,C 180,E1 -7849.615,E2 -7849.615} C_VEL
